LIN {X 0,Y 573.222,Z 156.084,A -85,B 0,C 180,E1 -2316.134,E2 -2316.134} C_VEL
LIN {X 0,Y 573.247,Z 156.08,A -85,B 0,C 180,E1 -2319.173,E2 -2319.173} C_VEL
LIN {X 0,Y 573.22,Z 156.083,A -85,B 0,C 180,E1 -2321.411,E2 -2321.411} C_VEL
LIN {X 0,Y 573.25,Z 156.076,A -85,B 0,C 180,E1 -2323.622,E2 -2323.622} C_VEL
LIN {X 0,Y 573.271,Z 156.075,A -85,B 0,C 180,E1 -2325.807,E2 -2325.807} C_VEL
LIN {X 0,Y 573.261,Z 156.075,A -85,B 0,C 180,E1 -2328.745,E2 -2328.745} C_VEL
LIN {X 0,Y 573.235,Z 156.083,A -85,B 0,C 180,E1 -2331.54,E2 -2331.54} C_VEL
LIN {X 0,Y 573.272,Z 156.074,A -85,B 0,C 180,E1 -2334.372,E2 -2334.372} C_VEL
LIN {X 0,Y 573.302,Z 156.07,A -85,B 0,C 180,E1 -2337.189,E2 -2337.189} C_VEL
LIN {X 0,Y 573.322,Z 156.073,A -85,B 0,C 180,E1 -2340,E2 -2340} C_VEL
LIN {X 0,Y 573.302,Z 156.07,A -85,B 0,C 180,E1 -2342.811,E2 -2342.811} C_VEL
LIN {X 0,Y 573.269,Z 156.075,A -85,B 0,C 180,E1 -2345.628,E2 -2345.628} C_VEL
LIN {X 0,Y 573.236,Z 156.083,A -85,B 0,C 180,E1 -2348.46,E2 -2348.46} C_VEL
LIN {X 0,Y 573.27,Z 156.073,A -85,B 0,C 180,E1 -2351.312,E2 -2351.312} C_VEL
LIN {X 0,Y 573.271,Z 156.075,A -85,B 0,C 180,E1 -2354.193,E2 -2354.193} C_VEL
LIN {X 0,Y 573.257,Z 156.081,A -85,B 0,C 180,E1 -2357.112,E2 -2357.112} C_VEL
LIN {X 0,Y 573.237,Z 156.079,A -85,B 0,C 180,E1 -2360.077,E2 -2360.077} C_VEL
LIN {X 0,Y 573.217,Z 156.086,A -85,B 0,C 180,E1 -2362.339,E2 -2362.339} C_VEL
LIN {X 0,Y 573.243,Z 156.077,A -85,B 0,C 180,E1 -2364.375,E2 -2364.375} C_VEL
LIN {X 0,Y 572.619,Z 156.154,A -85,B 0,C 180,E1 -2364.962,E2 -2364.962} C_VEL
LIN {X 0,Y 569.78,Z 156.514,A -85,B 0,C 180,E1 -2365.913,E2 -2365.913} C_VEL
LIN {X 0,Y 567.348,Z 156.82,A -85,B 0,C 180,E1 -2366.679,E2 -2366.679} C_VEL
LIN {X 0,Y 566.293,Z 156.949,A -85,B 0,C 180,E1 -2367.27,E2 -2367.27} C_VEL
LIN {X 0,Y 566.202,Z 156.958,A -85,B 0,C 180,E1 -2367.47,E2 -2367.47} C_VEL
LIN {X 0,Y 566.2,Z 156.955,A -85,B 0,C 180,E1 -2369.769,E2 -2369.769} C_VEL
LIN {X 0,Y 566.203,Z 156.96,A -85,B 0,C 180,E1 -2372.43,E2 -2372.43} C_VEL
LIN {X 0,Y 566.167,Z 156.959,A -85,B 0,C 180,E1 -2374.988,E2 -2374.988} C_VEL
LIN {X 0,Y 566.183,Z 156.961,A -85,B 0,C 180,E1 -2377.462,E2 -2377.462} C_VEL
LIN {X 0,Y 566.205,Z 156.953,A -85,B 0,C 180,E1 -2380.2,E2 -2380.2} C_VEL
LIN {X 0,Y 566.199,Z 156.958,A -85,B 0,C 180,E1 -2383.055,E2 -2383.055} C_VEL
LIN {X 0,Y 566.198,Z 156.959,A -85,B 0,C 180,E1 -2386.049,E2 -2386.049} C_VEL
LIN {X 0,Y 566.203,Z 156.956,A -85,B 0,C 180,E1 -2389.215,E2 -2389.215} C_VEL
LIN {X 0,Y 566.171,Z 156.962,A -85,B 0,C 180,E1 -2391.636,E2 -2391.636} C_VEL
LIN {X 0,Y 566.131,Z 156.965,A -85,B 0,C 180,E1 -2394.306,E2 -2394.306} C_VEL
LIN {X 0,Y 566.142,Z 157.825,A -85,B 0,C 180,E1 -2395.178,E2 -2395.178} C_VEL
LIN {X 0,Y 566.126,Z 162.015,A -85,B 0,C 180,E1 -2397.737,E2 -2397.737} C_VEL
LIN {X 0,Y 566.1,Z 166.291,A -85,B 0,C 180,E1 -2400.347,E2 -2400.347} C_VEL
LIN {X 0,Y 566.065,Z 170.142,A -85,B 0,C 180,E1 -2402.654,E2 -2402.654} C_VEL
LIN {X 0,Y 566.061,Z 174.191,A -85,B 0,C 180,E1 -2405.031,E2 -2405.031} C_VEL
LIN {X 0,Y 565.989,Z 178.243,A -85,B 0,C 180,E1 -2407.361,E2 -2407.361} C_VEL
LIN {X 0,Y 565.961,Z 182.275,A -85,B 0,C 180,E1 -2409.654,E2 -2409.654} C_VEL
LIN {X 0,Y 565.898,Z 186.291,A -85,B 0,C 180,E1 -2411.912,E2 -2411.912} C_VEL
LIN {X 0,Y 565.902,Z 191.779,A -85,B 0,C 180,E1 -2414.883,E2 -2414.883} C_VEL
LIN {X 0,Y 565.886,Z 196.532,A -85,B 0,C 180,E1 -2417.402,E2 -2417.402} C_VEL
LIN {X 0,Y 566.916,Z 203.459,A -85,B 0,C 180,E1 -2417.584,E2 -2417.584} C_VEL
LIN {X 0,Y 566.783,Z 216.489,A -85,B 0,C 180,E1 -2417.968,E2 -2417.968} C_VEL
LIN {X 0,Y 566.608,Z 229.064,A -85,B 0,C 180,E1 -2418.49,E2 -2418.49} C_VEL
LIN {X 0,Y 566.519,Z 240.338,A -85,B 0,C 180,E1 -2419.114,E2 -2419.114} C_VEL
LIN {X 0,Y 566.397,Z 251.686,A -85,B 0,C 180,E1 -2419.906,E2 -2419.906} C_VEL
LIN {X 0,Y 566.255,Z 261.061,A -85,B 0,C 180,E1 -2420.715,E2 -2420.715} C_VEL
LIN {X 0,Y 566.158,Z 269.617,A -85,B 0,C 180,E1 -2421.613,E2 -2421.613} C_VEL
LIN {X 0,Y 566.063,Z 277.929,A -85,B 0,C 180,E1 -2422.689,E2 -2422.689} C_VEL
LIN {X 0,Y 565.988,Z 284.624,A -85,B 0,C 180,E1 -2423.763,E2 -2423.763} C_VEL
LIN {X 0,Y 565.877,Z 290.765,A -85,B 0,C 180,E1 -2425.013,E2 -2425.013} C_VEL
LIN {X 0,Y 565.926,Z 294.754,A -85,B 0,C 180,E1 -2426.084,E2 -2426.084} C_VEL
LIN {X 0,Y 565.877,Z 297.703,A -85,B 0,C 180,E1 -2427.153,E2 -2427.153} C_VEL
LIN {X 0,Y 565.841,Z 299.128,A -85,B 0,C 180,E1 -2427.865,E2 -2427.865} C_VEL
LIN {X 0,Y 565.841,Z 300.756,A -85,B 0,C 180,E1 -2429.289,E2 -2429.289} C_VEL
LIN {X 0,Y 565.839,Z 300.996,A -85,B 0,C 180,E1 -2430,E2 -2430} C_VEL
LIN {X 0,Y 565.841,Z 300.815,A -85,B 0,C 180,E1 -2430.712,E2 -2430.712} C_VEL
LIN {X 0,Y 565.841,Z 299.267,A -85,B 0,C 180,E1 -2432.136,E2 -2432.136} C_VEL
LIN {X 0,Y 565.878,Z 297.906,A -85,B 0,C 180,E1 -2432.848,E2 -2432.848} C_VEL
LIN {X 0,Y 565.926,Z 295.029,A -85,B 0,C 180,E1 -2433.917,E2 -2433.917} C_VEL
LIN {X 0,Y 565.878,Z 291.128,A -85,B 0,C 180,E1 -2434.988,E2 -2434.988} C_VEL
LIN {X 0,Y 565.991,Z 286.096,A -85,B 0,C 180,E1 -2436.059,E2 -2436.059} C_VEL
LIN {X 0,Y 566.031,Z 279.771,A -85,B 0,C 180,E1 -2437.133,E2 -2437.133} C_VEL
LIN {X 0,Y 566.128,Z 271.849,A -85,B 0,C 180,E1 -2438.208,E2 -2438.208} C_VEL
LIN {X 0,Y 566.249,Z 261.997,A -85,B 0,C 180,E1 -2439.285,E2 -2439.285} C_VEL
LIN {X 0,Y 566.401,Z 251.679,A -85,B 0,C 180,E1 -2440.185,E2 -2440.185} C_VEL
LIN {X 0,Y 566.499,Z 240.539,A -85,B 0,C 180,E1 -2440.964,E2 -2440.964} C_VEL
LIN {X 0,Y 566.63,Z 229.184,A -85,B 0,C 180,E1 -2441.593,E2 -2441.593} C_VEL
LIN {X 0,Y 566.8,Z 216.59,A -85,B 0,C 180,E1 -2442.119,E2 -2442.119} C_VEL
LIN {X 0,Y 566.924,Z 203.412,A -85,B 0,C 180,E1 -2442.507,E2 -2442.507} C_VEL
LIN {X 0,Y 565.888,Z 196.529,A -85,B 0,C 180,E1 -2442.69,E2 -2442.69} C_VEL
LIN {X 0,Y 565.893,Z 191.947,A -85,B 0,C 180,E1 -2445.118,E2 -2445.118} C_VEL
LIN {X 0,Y 565.896,Z 186.449,A -85,B 0,C 180,E1 -2448.088,E2 -2448.088} C_VEL
LIN {X 0,Y 565.96,Z 182.428,A -85,B 0,C 180,E1 -2450.347,E2 -2450.347} C_VEL
LIN {X 0,Y 566.015,Z 177.311,A -85,B 0,C 180,E1 -2453.244,E2 -2453.244} C_VEL
LIN {X 0,Y 566.035,Z 173,A -85,B 0,C 180,E1 -2455.758,E2 -2455.758} C_VEL
LIN {X 0,Y 566.085,Z 168.894,A -85,B 0,C 180,E1 -2458.179,E2 -2458.179} C_VEL
LIN {X 0,Y 566.108,Z 164.128,A -85,B 0,C 180,E1 -2461.062,E2 -2461.062} C_VEL
LIN {X 0,Y 566.151,Z 159.371,A -85,B 0,C 180,E1 -2463.96,E2 -2463.96} C_VEL
LIN {X 0,Y 566.159,Z 157.704,A -85,B 0,C 180,E1 -2464.986,E2 -2464.986} C_VEL
LIN {X 0,Y 566.115,Z 156.967,A -85,B 0,C 180,E1 -2465.696,E2 -2465.696} C_VEL
LIN {X 0,Y 566.182,Z 156.962,A -85,B 0,C 180,E1 -2468.554,E2 -2468.554} C_VEL
LIN {X 0,Y 566.161,Z 156.959,A -85,B 0,C 180,E1 -2471.141,E2 -2471.141} C_VEL
LIN {X 0,Y 566.199,Z 156.959,A -85,B 0,C 180,E1 -2474.036,E2 -2474.036} C_VEL
LIN {X 0,Y 566.203,Z 156.958,A -85,B 0,C 180,E1 -2477.083,E2 -2477.083} C_VEL
LIN {X 0,Y 566.214,Z 156.954,A -85,B 0,C 180,E1 -2480.314,E2 -2480.314} C_VEL
LIN {X 0,Y 566.186,Z 156.96,A -85,B 0,C 180,E1 -2482.601,E2 -2482.601} C_VEL
LIN {X 0,Y 566.183,Z 156.957,A -85,B 0,C 180,E1 -2485.18,E2 -2485.18} C_VEL
LIN {X 0,Y 566.232,Z 156.955,A -85,B 0,C 180,E1 -2487.743,E2 -2487.743} C_VEL
LIN {X 0,Y 566.205,Z 156.954,A -85,B 0,C 180,E1 -2490.328,E2 -2490.328} C_VEL
LIN {X 0,Y 566.212,Z 156.959,A -85,B 0,C 180,E1 -2492.661,E2 -2492.661} C_VEL
LIN {X 0,Y 566.238,Z 156.949,A -85,B 0,C 180,E1 -2495.039,E2 -2495.039} C_VEL
LIN {X 0,Y 566.185,Z 156.959,A -85,B 0,C 180,E1 -2498.137,E2 -2498.137} C_VEL
LIN {X 0,Y 566.231,Z 156.951,A -85,B 0,C 180,E1 -2500.614,E2 -2500.614} C_VEL
LIN {X 0,Y 566.216,Z 156.954,A -85,B 0,C 180,E1 -2503.412,E2 -2503.412} C_VEL
LIN {X 0,Y 566.198,Z 156.961,A -85,B 0,C 180,E1 -2506.359,E2 -2506.359} C_VEL
LIN {X 0,Y 566.236,Z 156.95,A -85,B 0,C 180,E1 -2508.675,E2 -2508.675} C_VEL
LIN {X 0,Y 566.193,Z 156.961,A -85,B 0,C 180,E1 -2511.434,E2 -2511.434} C_VEL
LIN {X 0,Y 566.233,Z 156.95,A -85,B 0,C 180,E1 -2514.301,E2 -2514.301} C_VEL
LIN {X 0,Y 566.269,Z 156.947,A -85,B 0,C 180,E1 -2517.154,E2 -2517.154} C_VEL
LIN {X 0,Y 566.293,Z 156.949,A -85,B 0,C 180,E1 -2520,E2 -2520} C_VEL
LIN {X 0,Y 566.271,Z 156.946,A -85,B 0,C 180,E1 -2522.846,E2 -2522.846} C_VEL
LIN {X 0,Y 566.241,Z 156.95,A -85,B 0,C 180,E1 -2525.698,E2 -2525.698} C_VEL
LIN {X 0,Y 566.189,Z 156.961,A -85,B 0,C 180,E1 -2528.566,E2 -2528.566} C_VEL
LIN {X 0,Y 566.243,Z 156.95,A -85,B 0,C 180,E1 -2531.454,E2 -2531.454} C_VEL
LIN {X 0,Y 566.236,Z 156.95,A -85,B 0,C 180,E1 -2534.507,E2 -2534.507} C_VEL
LIN {X 0,Y 566.2,Z 156.96,A -85,B 0,C 180,E1 -2537.332,E2 -2537.332} C_VEL
LIN {X 0,Y 566.206,Z 156.957,A -85,B 0,C 180,E1 -2540.337,E2 -2540.337} C_VEL
LIN {X 0,Y 566.166,Z 156.958,A -85,B 0,C 180,E1 -2543.28,E2 -2543.28} C_VEL
LIN {X 0,Y 566.207,Z 156.96,A -85,B 0,C 180,E1 -2545.749,E2 -2545.749} C_VEL
LIN {X 0,Y 566.204,Z 156.954,A -85,B 0,C 180,E1 -2548.202,E2 -2548.202} C_VEL
LIN {X 0,Y 566.193,Z 156.96,A -85,B 0,C 180,E1 -2551.077,E2 -2551.077} C_VEL
LIN {X 0,Y 566.212,Z 156.954,A -85,B 0,C 180,E1 -2553.734,E2 -2553.734} C_VEL
LIN {X 0,Y 566.145,Z 156.962,A -85,B 0,C 180,E1 -2556.574,E2 -2556.574} C_VEL
LIN {X 0,Y 566.205,Z 156.958,A -85,B 0,C 180,E1 -2559.275,E2 -2559.275} C_VEL
LIN {X 0,Y 566.19,Z 156.955,A -85,B 0,C 180,E1 -2562.09,E2 -2562.09} C_VEL
LIN {X 0,Y 566.17,Z 156.96,A -85,B 0,C 180,E1 -2565.036,E2 -2565.036} C_VEL
LIN {X 0,Y 566.19,Z 156.961,A -85,B 0,C 180,E1 -2567.91,E2 -2567.91} C_VEL
LIN {X 0,Y 566.206,Z 156.955,A -85,B 0,C 180,E1 -2570.726,E2 -2570.726} C_VEL
LIN {X 0,Y 566.203,Z 157.05,A -85,B 0,C 180,E1 -2573.481,E2 -2573.481} C_VEL
LIN {X 0,Y 566.594,Z 160.732,A -85,B 0,C 180,E1 -2574.951,E2 -2574.951} C_VEL
LIN {X 0,Y 566.468,Z 168.073,A -85,B 0,C 180,E1 -2577.759,E2 -2577.759} C_VEL
LIN {X 0,Y 566.419,Z 174.878,A -85,B 0,C 180,E1 -2580.29,E2 -2580.29} C_VEL
LIN {X 0,Y 566.308,Z 183.258,A -85,B 0,C 180,E1 -2583.321,E2 -2583.321} C_VEL
LIN {X 0,Y 566.224,Z 191.447,A -85,B 0,C 180,E1 -2586.21,E2 -2586.21} C_VEL
LIN {X 0,Y 566.162,Z 199.239,A -85,B 0,C 180,E1 -2588.9,E2 -2588.9} C_VEL
LIN {X 0,Y 566.083,Z 207.03,A -85,B 0,C 180,E1 -2591.543,E2 -2591.543} C_VEL
LIN {X 0,Y 566.024,Z 215.935,A -85,B 0,C 180,E1 -2594.517,E2 -2594.517} C_VEL
LIN {X 0,Y 565.976,Z 224.283,A -85,B 0,C 180,E1 -2597.267,E2 -2597.267} C_VEL
LIN {X 0,Y 565.964,Z 224.491,A -85,B 0,C 180,E1 -2597.335,E2 -2597.335} C_VEL
LIN {X 0,Y 566.944,Z 231.504,A -85,B 0,C 180,E1 -2597.494,E2 -2597.494} C_VEL
LIN {X 0,Y 566.824,Z 243.874,A -85,B 0,C 180,E1 -2597.832,E2 -2597.832} C_VEL
LIN {X 0,Y 566.64,Z 256.897,A -85,B 0,C 180,E1 -2598.346,E2 -2598.346} C_VEL
LIN {X 0,Y 566.528,Z 268.482,A -85,B 0,C 180,E1 -2598.955,E2 -2598.955} C_VEL
LIN {X 0,Y 566.432,Z 279.927,A -85,B 0,C 180,E1 -2599.726,E2 -2599.726} C_VEL
LIN {X 0,Y 566.282,Z 289.599,A -85,B 0,C 180,E1 -2600.535,E2 -2600.535} C_VEL
LIN {X 0,Y 566.181,Z 298.412,A -85,B 0,C 180,E1 -2601.433,E2 -2601.433} C_VEL
LIN {X 0,Y 566.056,Z 306.999,A -85,B 0,C 180,E1 -2602.509,E2 -2602.509} C_VEL
LIN {X 0,Y 565.965,Z 313.866,A -85,B 0,C 180,E1 -2603.583,E2 -2603.583} C_VEL
LIN {X 0,Y 565.937,Z 319.365,A -85,B 0,C 180,E1 -2604.656,E2 -2604.656} C_VEL
LIN {X 0,Y 565.959,Z 323.677,A -85,B 0,C 180,E1 -2605.727,E2 -2605.727} C_VEL
LIN {X 0,Y 565.927,Z 325.956,A -85,B 0,C 180,E1 -2606.44,E2 -2606.44} C_VEL
LIN {X 0,Y 565.878,Z 327.808,A -85,B 0,C 180,E1 -2607.152,E2 -2607.152} C_VEL
LIN {X 0,Y 565.841,Z 329.2,A -85,B 0,C 180,E1 -2607.864,E2 -2607.864} C_VEL
LIN {X 0,Y 565.841,Z 330.784,A -85,B 0,C 180,E1 -2609.288,E2 -2609.288} C_VEL
LIN {X 0,Y 565.839,Z 331,A -85,B 0,C 180,E1 -2610,E2 -2610} C_VEL
LIN {X 0,Y 565.846,Z 330.186,A -85,B 0,C 180,E1 -2611.423,E2 -2611.423} C_VEL
LIN {X 0,Y 565.841,Z 329.201,A -85,B 0,C 180,E1 -2612.135,E2 -2612.135} C_VEL
LIN {X 0,Y 565.878,Z 327.81,A -85,B 0,C 180,E1 -2612.847,E2 -2612.847} C_VEL
LIN {X 0,Y 565.926,Z 324.897,A -85,B 0,C 180,E1 -2613.916,E2 -2613.916} C_VEL
LIN {X 0,Y 565.878,Z 320.95,A -85,B 0,C 180,E1 -2614.987,E2 -2614.987} C_VEL
LIN {X 0,Y 566.002,Z 315.867,A -85,B 0,C 180,E1 -2616.058,E2 -2616.058} C_VEL
LIN {X 0,Y 566.04,Z 309.471,A -85,B 0,C 180,E1 -2617.132,E2 -2617.132} C_VEL
LIN {X 0,Y 566.133,Z 301.48,A -85,B 0,C 180,E1 -2618.207,E2 -2618.207} C_VEL
LIN {X 0,Y 566.229,Z 293.339,A -85,B 0,C 180,E1 -2619.105,E2 -2619.105} C_VEL
LIN {X 0,Y 566.336,Z 283.405,A -85,B 0,C 180,E1 -2620.005,E2 -2620.005} C_VEL
LIN {X 0,Y 566.469,Z 272.332,A -85,B 0,C 180,E1 -2620.805,E2 -2620.805} C_VEL
LIN {X 0,Y 566.608,Z 259.955,A -85,B 0,C 180,E1 -2621.51,E2 -2621.51} C_VEL
LIN {X 0,Y 566.746,Z 247.773,A -85,B 0,C 180,E1 -2622.033,E2 -2622.033} C_VEL
LIN {X 0,Y 566.906,Z 234.359,A -85,B 0,C 180,E1 -2622.439,E2 -2622.439} C_VEL
LIN {X 0,Y 566.632,Z 228.828,A -85,B 0,C 180,E1 -2622.567,E2 -2622.567} C_VEL
LIN {X 0,Y 565.963,Z 224.492,A -85,B 0,C 180,E1 -2622.665,E2 -2622.665} C_VEL
LIN {X 0,Y 566.019,Z 217.049,A -85,B 0,C 180,E1 -2625.114,E2 -2625.114} C_VEL
LIN {X 0,Y 566.065,Z 208.144,A -85,B 0,C 180,E1 -2628.082,E2 -2628.082} C_VEL
LIN {X 0,Y 566.145,Z 200.353,A -85,B 0,C 180,E1 -2630.719,E2 -2630.719} C_VEL
LIN {X 0,Y 566.205,Z 192.562,A -85,B 0,C 180,E1 -2633.403,E2 -2633.403} C_VEL
LIN {X 0,Y 566.294,Z 184.77,A -85,B 0,C 180,E1 -2636.14,E2 -2636.14} C_VEL
LIN {X 0,Y 566.383,Z 176.979,A -85,B 0,C 180,E1 -2638.942,E2 -2638.942} C_VEL
LIN {X 0,Y 566.477,Z 169.187,A -85,B 0,C 180,E1 -2641.821,E2 -2641.821} C_VEL
LIN {X 0,Y 566.567,Z 161.396,A -85,B 0,C 180,E1 -2644.792,E2 -2644.792} C_VEL
LIN {X 0,Y 566.225,Z 157.187,A -85,B 0,C 180,E1 -2646.466,E2 -2646.466} C_VEL
LIN {X 0,Y 566.201,Z 156.961,A -85,B 0,C 180,E1 -2646.569,E2 -2646.569} C_VEL
LIN {X 0,Y 566.208,Z 156.955,A -85,B 0,C 180,E1 -2649.685,E2 -2649.685} C_VEL
LIN {X 0,Y 566.208,Z 156.96,A -85,B 0,C 180,E1 -2652.087,E2 -2652.087} C_VEL
LIN {X 0,Y 566.168,Z 156.961,A -85,B 0,C 180,E1 -2655.036,E2 -2655.036} C_VEL
LIN {X 0,Y 566.188,Z 156.956,A -85,B 0,C 180,E1 -2657.91,E2 -2657.91} C_VEL
LIN {X 0,Y 566.206,Z 156.958,A -85,B 0,C 180,E1 -2660.725,E2 -2660.725} C_VEL
LIN {X 0,Y 566.143,Z 156.962,A -85,B 0,C 180,E1 -2663.426,E2 -2663.426} C_VEL
LIN {X 0,Y 566.209,Z 156.954,A -85,B 0,C 180,E1 -2666.266,E2 -2666.266} C_VEL
LIN {X 0,Y 566.194,Z 156.959,A -85,B 0,C 180,E1 -2668.922,E2 -2668.922} C_VEL
LIN {X 0,Y 566.21,Z 156.953,A -85,B 0,C 180,E1 -2671.857,E2 -2671.857} C_VEL
LIN {X 0,Y 566.211,Z 156.96,A -85,B 0,C 180,E1 -2674.251,E2 -2674.251} C_VEL
LIN {X 0,Y 566.164,Z 156.958,A -85,B 0,C 180,E1 -2676.72,E2 -2676.72} C_VEL
LIN {X 0,Y 566.204,Z 156.958,A -85,B 0,C 180,E1 -2679.662,E2 -2679.662} C_VEL
LIN {X 0,Y 566.198,Z 156.959,A -85,B 0,C 180,E1 -2682.668,E2 -2682.668} C_VEL
LIN {X 0,Y 566.232,Z 156.951,A -85,B 0,C 180,E1 -2685.627,E2 -2685.627} C_VEL
LIN {X 0,Y 566.232,Z 156.95,A -85,B 0,C 180,E1 -2688.675,E2 -2688.675} C_VEL
LIN {X 0,Y 566.189,Z 156.962,A -85,B 0,C 180,E1 -2691.434,E2 -2691.434} C_VEL
LIN {X 0,Y 566.238,Z 156.95,A -85,B 0,C 180,E1 -2694.301,E2 -2694.301} C_VEL
LIN {X 0,Y 566.275,Z 156.947,A -85,B 0,C 180,E1 -2697.866,E2 -2697.866} C_VEL
LIN {X 0,Y 566.301,Z 156.942,A -85,B 0,C 180,E1 -2700.711,E2 -2700.711} C_VEL
LIN {X 0,Y 566.269,Z 156.947,A -85,B 0,C 180,E1 -2702.846,E2 -2702.846} C_VEL
LIN {X 0,Y 566.236,Z 156.95,A -85,B 0,C 180,E1 -2705.699,E2 -2705.699} C_VEL
LIN {X 0,Y 566.19,Z 156.962,A -85,B 0,C 180,E1 -2708.566,E2 -2708.566} C_VEL
LIN {X 0,Y 566.24,Z 156.95,A -85,B 0,C 180,E1 -2711.454,E2 -2711.454} C_VEL
LIN {X 0,Y 566.233,Z 156.95,A -85,B 0,C 180,E1 -2714.507,E2 -2714.507} C_VEL
LIN {X 0,Y 566.198,Z 156.959,A -85,B 0,C 180,E1 -2717.332,E2 -2717.332} C_VEL
LIN {X 0,Y 566.203,Z 156.958,A -85,B 0,C 180,E1 -2720.338,E2 -2720.338} C_VEL
LIN {X 0,Y 566.164,Z 156.958,A -85,B 0,C 180,E1 -2723.28,E2 -2723.28} C_VEL
LIN {X 0,Y 566.211,Z 156.959,A -85,B 0,C 180,E1 -2725.749,E2 -2725.749} C_VEL
LIN {X 0,Y 566.202,Z 156.958,A -85,B 0,C 180,E1 -2727.47,E2 -2727.47} C_VEL
LIN {X 0,Y 565.521,Z 157.04,A -85,B 0,C 180,E1 -2728.064,E2 -2728.064} C_VEL
LIN {X 0,Y 562.656,Z 157.401,A -85,B 0,C 180,E1 -2729.027,E2 -2729.027} C_VEL
LIN {X 0,Y 560.247,Z 157.698,A -85,B 0,C 180,E1 -2729.803,E2 -2729.803} C_VEL
LIN {X 0,Y 559.22,Z 157.826,A -85,B 0,C 180,E1 -2730.402,E2 -2730.402} C_VEL
LIN {X 0,Y 559.139,Z 157.835,A -85,B 0,C 180,E1 -2730.604,E2 -2730.604} C_VEL
LIN {X 0,Y 559.156,Z 157.837,A -85,B 0,C 180,E1 -2732.715,E2 -2732.715} C_VEL
LIN {X 0,Y 559.115,Z 157.837,A -85,B 0,C 180,E1 -2735.325,E2 -2735.325} C_VEL
LIN {X 0,Y 559.121,Z 157.838,A -85,B 0,C 180,E1 -2738.019,E2 -2738.019} C_VEL
LIN {X 0,Y 559.155,Z 157.834,A -85,B 0,C 180,E1 -2740.813,E2 -2740.813} C_VEL
LIN {X 0,Y 559.138,Z 157.834,A -85,B 0,C 180,E1 -2743.734,E2 -2743.734} C_VEL
LIN {X 0,Y 559.146,Z 157.834,A -85,B 0,C 180,E1 -2746.804,E2 -2746.804} C_VEL
LIN {X 0,Y 559.155,Z 157.834,A -85,B 0,C 180,E1 -2749.188,E2 -2749.188} C_VEL
LIN {X 0,Y 559.121,Z 157.837,A -85,B 0,C 180,E1 -2751.982,E2 -2751.982} C_VEL
LIN {X 0,Y 559.054,Z 157.882,A -85,B 0,C 180,E1 -2754.671,E2 -2754.671} C_VEL
LIN {X 0,Y 559.057,Z 162.259,A -85,B 0,C 180,E1 -2757.381,E2 -2757.381} C_VEL
LIN {X 0,Y 559.053,Z 166.761,A -85,B 0,C 180,E1 -2760.16,E2 -2760.16} C_VEL
LIN {X 0,Y 558.994,Z 171.604,A -85,B 0,C 180,E1 -2763.089,E2 -2763.089} C_VEL
LIN {X 0,Y 558.955,Z 175.655,A -85,B 0,C 180,E1 -2765.486,E2 -2765.486} C_VEL
LIN {X 0,Y 558.929,Z 180.876,A -85,B 0,C 180,E1 -2768.51,E2 -2768.51} C_VEL
LIN {X 0,Y 558.89,Z 185.109,A -85,B 0,C 180,E1 -2770.917,E2 -2770.917} C_VEL
LIN {X 0,Y 558.788,Z 190.462,A -85,B 0,C 180,E1 -2773.937,E2 -2773.937} C_VEL
LIN {X 0,Y 558.781,Z 194.545,A -85,B 0,C 180,E1 -2776.174,E2 -2776.174} C_VEL
LIN {X 0,Y 558.817,Z 196.533,A -85,B 0,C 180,E1 -2777.24,E2 -2777.24} C_VEL
LIN {X 0,Y 560.002,Z 204.395,A -85,B 0,C 180,E1 -2777.451,E2 -2777.451} C_VEL
LIN {X 0,Y 559.846,Z 216.89,A -85,B 0,C 180,E1 -2777.83,E2 -2777.83} C_VEL
LIN {X 0,Y 559.665,Z 228.866,A -85,B 0,C 180,E1 -2778.335,E2 -2778.335} C_VEL
LIN {X 0,Y 559.531,Z 240.553,A -85,B 0,C 180,E1 -2778.989,E2 -2778.989} C_VEL
LIN {X 0,Y 559.393,Z 251.692,A -85,B 0,C 180,E1 -2779.778,E2 -2779.778} C_VEL
LIN {X 0,Y 559.239,Z 261.068,A -85,B 0,C 180,E1 -2780.598,E2 -2780.598} C_VEL
LIN {X 0,Y 559.129,Z 269.623,A -85,B 0,C 180,E1 -2781.507,E2 -2781.507} C_VEL
LIN {X 0,Y 558.988,Z 277.932,A -85,B 0,C 180,E1 -2782.596,E2 -2782.596} C_VEL
LIN {X 0,Y 558.89,Z 284.414,A -85,B 0,C 180,E1 -2783.645,E2 -2783.645} C_VEL
LIN {X 0,Y 558.869,Z 289.165,A -85,B 0,C 180,E1 -2784.588,E2 -2784.588} C_VEL
LIN {X 0,Y 558.868,Z 293.523,A -85,B 0,C 180,E1 -2785.673,E2 -2785.673} C_VEL
LIN {X 0,Y 558.836,Z 295.829,A -85,B 0,C 180,E1 -2786.395,E2 -2786.395} C_VEL
LIN {X 0,Y 558.799,Z 297.705,A -85,B 0,C 180,E1 -2787.117,E2 -2787.117} C_VEL
LIN {X 0,Y 558.747,Z 299.128,A -85,B 0,C 180,E1 -2787.838,E2 -2787.838} C_VEL
LIN {X 0,Y 558.741,Z 300.757,A -85,B 0,C 180,E1 -2789.279,E2 -2789.279} C_VEL
LIN {X 0,Y 558.74,Z 300.996,A -85,B 0,C 180,E1 -2790,E2 -2790} C_VEL
LIN {X 0,Y 558.741,Z 300.815,A -85,B 0,C 180,E1 -2790.721,E2 -2790.721} C_VEL
LIN {X 0,Y 558.747,Z 299.265,A -85,B 0,C 180,E1 -2792.163,E2 -2792.163} C_VEL
LIN {X 0,Y 558.8,Z 297.904,A -85,B 0,C 180,E1 -2792.884,E2 -2792.884} C_VEL
LIN {X 0,Y 558.844,Z 295.027,A -85,B 0,C 180,E1 -2793.966,E2 -2793.966} C_VEL
LIN {X 0,Y 558.798,Z 291.126,A -85,B 0,C 180,E1 -2795.051,E2 -2795.051} C_VEL
LIN {X 0,Y 558.911,Z 286.094,A -85,B 0,C 180,E1 -2796.136,E2 -2796.136} C_VEL
LIN {X 0,Y 558.973,Z 279.767,A -85,B 0,C 180,E1 -2797.223,E2 -2797.223} C_VEL
LIN {X 0,Y 559.091,Z 271.844,A -85,B 0,C 180,E1 -2798.312,E2 -2798.312} C_VEL
LIN {X 0,Y 559.223,Z 261.99,A -85,B 0,C 180,E1 -2799.403,E2 -2799.403} C_VEL
LIN {X 0,Y 559.399,Z 251.669,A -85,B 0,C 180,E1 -2800.313,E2 -2800.313} C_VEL
LIN {X 0,Y 559.504,Z 240.822,A -85,B 0,C 180,E1 -2801.084,E2 -2801.084} C_VEL
LIN {X 0,Y 559.639,Z 230.269,A -85,B 0,C 180,E1 -2801.683,E2 -2801.683} C_VEL
LIN {X 0,Y 559.838,Z 217.741,A -85,B 0,C 180,E1 -2802.23,E2 -2802.23} C_VEL
LIN {X 0,Y 559.988,Z 204.304,A -85,B 0,C 180,E1 -2802.641,E2 -2802.641} C_VEL
LIN {X 0,Y 558.786,Z 196.528,A -85,B 0,C 180,E1 -2802.854,E2 -2802.854} C_VEL
LIN {X 0,Y 558.812,Z 191.964,A -85,B 0,C 180,E1 -2805.314,E2 -2805.314} C_VEL
LIN {X 0,Y 558.825,Z 186.593,A -85,B 0,C 180,E1 -2808.325,E2 -2808.325} C_VEL
LIN {X 0,Y 558.882,Z 182.561,A -85,B 0,C 180,E1 -2810.616,E2 -2810.616} C_VEL
LIN {X 0,Y 558.942,Z 177.747,A -85,B 0,C 180,E1 -2813.381,E2 -2813.381} C_VEL
LIN {X 0,Y 558.966,Z 173.106,A -85,B 0,C 180,E1 -2816.108,E2 -2816.108} C_VEL
LIN {X 0,Y 559.035,Z 169.048,A -85,B 0,C 180,E1 -2818.537,E2 -2818.537} C_VEL
LIN {X 0,Y 559.072,Z 164.601,A -85,B 0,C 180,E1 -2821.26,E2 -2821.26} C_VEL
LIN {X 0,Y 559.107,Z 159.435,A -85,B 0,C 180,E1 -2824.448,E2 -2824.448} C_VEL
LIN {X 0,Y 559.08,Z 158.027,A -85,B 0,C 180,E1 -2825.328,E2 -2825.328} C_VEL
LIN {X 0,Y 559.118,Z 157.837,A -85,B 0,C 180,E1 -2827.637,E2 -2827.637} C_VEL
LIN {X 0,Y 559.157,Z 157.833,A -85,B 0,C 180,E1 -2829.941,E2 -2829.941} C_VEL
LIN {X 0,Y 559.158,Z 157.832,A -85,B 0,C 180,E1 -2832.744,E2 -2832.744} C_VEL
LIN {X 0,Y 559.151,Z 157.836,A -85,B 0,C 180,E1 -2835.761,E2 -2835.761} C_VEL
LIN {X 0,Y 559.164,Z 157.83,A -85,B 0,C 180,E1 -2838.23,E2 -2838.23} C_VEL
LIN {X 0,Y 559.171,Z 157.831,A -85,B 0,C 180,E1 -2841.192,E2 -2841.192} C_VEL
LIN {X 0,Y 559.115,Z 157.84,A -85,B 0,C 180,E1 -2843.787,E2 -2843.787} C_VEL
LIN {X 0,Y 559.146,Z 157.834,A -85,B 0,C 180,E1 -2846.424,E2 -2846.424} C_VEL
LIN {X 0,Y 559.157,Z 157.836,A -85,B 0,C 180,E1 -2848.981,E2 -2848.981} C_VEL
LIN {X 0,Y 559.17,Z 157.83,A -85,B 0,C 180,E1 -2851.619,E2 -2851.619} C_VEL
LIN {X 0,Y 559.182,Z 157.829,A -85,B 0,C 180,E1 -2853.903,E2 -2853.903} C_VEL
LIN {X 0,Y 559.137,Z 157.835,A -85,B 0,C 180,E1 -2856.572,E2 -2856.572} C_VEL
LIN {X 0,Y 559.174,Z 157.834,A -85,B 0,C 180,E1 -2859.395,E2 -2859.395} C_VEL
LIN {X 0,Y 559.139,Z 157.836,A -85,B 0,C 180,E1 -2861.685,E2 -2861.685} C_VEL
LIN {X 0,Y 559.167,Z 157.831,A -85,B 0,C 180,E1 -2863.948,E2 -2863.948} C_VEL
LIN {X 0,Y 559.173,Z 157.835,A -85,B 0,C 180,E1 -2866.184,E2 -2866.184} C_VEL
LIN {X 0,Y 559.194,Z 157.827,A -85,B 0,C 180,E1 -2869.133,E2 -2869.133} C_VEL
LIN {X 0,Y 559.138,Z 157.834,A -85,B 0,C 180,E1 -2872.053,E2 -2872.053} C_VEL
LIN {X 0,Y 559.24,Z 157.827,A -85,B 0,C 180,E1 -2874.953,E2 -2874.953} C_VEL
LIN {X 0,Y 559.245,Z 157.822,A -85,B 0,C 180,E1 -2877.839,E2 -2877.839} C_VEL
LIN {X 0,Y 559.274,Z 157.818,A -85,B 0,C 180,E1 -2880.72,E2 -2880.72} C_VEL
LIN {X 0,Y 559.237,Z 157.822,A -85,B 0,C 180,E1 -2882.881,E2 -2882.881} C_VEL
LIN {X 0,Y 559.209,Z 157.825,A -85,B 0,C 180,E1 -2885.77,E2 -2885.77} C_VEL
LIN {X 0,Y 559.156,Z 157.838,A -85,B 0,C 180,E1 -2888.675,E2 -2888.675} C_VEL
LIN {X 0,Y 559.206,Z 157.827,A -85,B 0,C 180,E1 -2891.6,E2 -2891.6} C_VEL
LIN {X 0,Y 559.202,Z 157.826,A -85,B 0,C 180,E1 -2894.596,E2 -2894.596} C_VEL
LIN {X 0,Y 559.143,Z 157.836,A -85,B 0,C 180,E1 -2897.557,E2 -2897.557} C_VEL
LIN {X 0,Y 559.166,Z 157.83,A -85,B 0,C 180,E1 -2899.838,E2 -2899.838} C_VEL
LIN {X 0,Y 559.137,Z 157.839,A -85,B 0,C 180,E1 -2902.153,E2 -2902.153} C_VEL
LIN {X 0,Y 559.175,Z 157.831,A -85,B 0,C 180,E1 -2905.298,E2 -2905.298} C_VEL
LIN {X 0,Y 559.169,Z 157.83,A -85,B 0,C 180,E1 -2908.381,E2 -2908.381} C_VEL
LIN {X 0,Y 559.148,Z 157.835,A -85,B 0,C 180,E1 -2911.273,E2 -2911.273} C_VEL
LIN {X 0,Y 559.165,Z 157.833,A -85,B 0,C 180,E1 -2913.949,E2 -2913.949} C_VEL
LIN {X 0,Y 559.112,Z 157.837,A -85,B 0,C 180,E1 -2917.111,E2 -2917.111} C_VEL
LIN {X 0,Y 559.157,Z 157.832,A -85,B 0,C 180,E1 -2919.941,E2 -2919.941} C_VEL
LIN {X 0,Y 559.158,Z 157.836,A -85,B 0,C 180,E1 -2922.744,E2 -2922.744} C_VEL
LIN {X 0,Y 559.151,Z 157.834,A -85,B 0,C 180,E1 -2925.761,E2 -2925.761} C_VEL
LIN {X 0,Y 559.164,Z 157.835,A -85,B 0,C 180,E1 -2928.23,E2 -2928.23} C_VEL
LIN {X 0,Y 559.168,Z 157.836,A -85,B 0,C 180,E1 -2931.193,E2 -2931.193} C_VEL
LIN {X 0,Y 559.19,Z 157.999,A -85,B 0,C 180,E1 -2933.341,E2 -2933.341} C_VEL
LIN {X 0,Y 559.588,Z 162.52,A -85,B 0,C 180,E1 -2935.155,E2 -2935.155} C_VEL
LIN {X 0,Y 559.47,Z 170.299,A -85,B 0,C 180,E1 -2938.157,E2 -2938.157} C_VEL
LIN {X 0,Y 559.428,Z 176.978,A -85,B 0,C 180,E1 -2940.663,E2 -2940.663} C_VEL
LIN {X 0,Y 559.275,Z 184.835,A -85,B 0,C 180,E1 -2943.53,E2 -2943.53} C_VEL
LIN {X 0,Y 559.167,Z 193.358,A -85,B 0,C 180,E1 -2946.566,E2 -2946.566} C_VEL
LIN {X 0,Y 559.097,Z 201.465,A -85,B 0,C 180,E1 -2949.392,E2 -2949.392} C_VEL
LIN {X 0,Y 559.01,Z 209.256,A -85,B 0,C 180,E1 -2952.06,E2 -2952.06} C_VEL
LIN {X 0,Y 558.943,Z 217.048,A -85,B 0,C 180,E1 -2954.689,E2 -2954.689} C_VEL
LIN {X 0,Y 558.906,Z 224.491,A -85,B 0,C 180,E1 -2957.172,E2 -2957.172} C_VEL
LIN {X 0,Y 560.004,Z 232.518,A -85,B 0,C 180,E1 -2957.359,E2 -2957.359} C_VEL
LIN {X 0,Y 559.883,Z 245.304,A -85,B 0,C 180,E1 -2957.729,E2 -2957.729} C_VEL
LIN {X 0,Y 559.682,Z 258.23,A -85,B 0,C 180,E1 -2958.261,E2 -2958.261} C_VEL
LIN {X 0,Y 559.549,Z 268.95,A -85,B 0,C 180,E1 -2958.843,E2 -2958.843} C_VEL
LIN {X 0,Y 559.42,Z 279.926,A -85,B 0,C 180,E1 -2959.596,E2 -2959.596} C_VEL
LIN {X 0,Y 559.243,Z 289.599,A -85,B 0,C 180,E1 -2960.415,E2 -2960.415} C_VEL
LIN {X 0,Y 559.127,Z 298.412,A -85,B 0,C 180,E1 -2961.325,E2 -2961.325} C_VEL
LIN {X 0,Y 558.996,Z 306.999,A -85,B 0,C 180,E1 -2962.414,E2 -2962.414} C_VEL
LIN {X 0,Y 558.885,Z 314.687,A -85,B 0,C 180,E1 -2963.649,E2 -2963.649} C_VEL
LIN {X 0,Y 558.869,Z 319.365,A -85,B 0,C 180,E1 -2964.588,E2 -2964.588} C_VEL
LIN {X 0,Y 558.868,Z 323.677,A -85,B 0,C 180,E1 -2965.673,E2 -2965.673} C_VEL
LIN {X 0,Y 558.836,Z 325.956,A -85,B 0,C 180,E1 -2966.395,E2 -2966.395} C_VEL
LIN {X 0,Y 558.799,Z 327.808,A -85,B 0,C 180,E1 -2967.116,E2 -2967.116} C_VEL
LIN {X 0,Y 558.746,Z 329.199,A -85,B 0,C 180,E1 -2967.837,E2 -2967.837} C_VEL
LIN {X 0,Y 558.741,Z 330.784,A -85,B 0,C 180,E1 -2969.279,E2 -2969.279} C_VEL
LIN {X 0,Y 558.74,Z 331,A -85,B 0,C 180,E1 -2970,E2 -2970} C_VEL
LIN {X 0,Y 558.745,Z 330.186,A -85,B 0,C 180,E1 -2971.441,E2 -2971.441} C_VEL
LIN {X 0,Y 558.746,Z 329.201,A -85,B 0,C 180,E1 -2972.162,E2 -2972.162} C_VEL
LIN {X 0,Y 558.799,Z 327.81,A -85,B 0,C 180,E1 -2972.883,E2 -2972.883} C_VEL
LIN {X 0,Y 558.844,Z 324.896,A -85,B 0,C 180,E1 -2973.966,E2 -2973.966} C_VEL
LIN {X 0,Y 558.798,Z 320.95,A -85,B 0,C 180,E1 -2975.051,E2 -2975.051} C_VEL
LIN {X 0,Y 558.921,Z 315.867,A -85,B 0,C 180,E1 -2976.135,E2 -2976.135} C_VEL
LIN {X 0,Y 558.977,Z 309.471,A -85,B 0,C 180,E1 -2977.223,E2 -2977.223} C_VEL
LIN {X 0,Y 559.099,Z 301.48,A -85,B 0,C 180,E1 -2978.311,E2 -2978.311} C_VEL
LIN {X 0,Y 559.194,Z 293.339,A -85,B 0,C 180,E1 -2979.221,E2 -2979.221} C_VEL
LIN {X 0,Y 559.346,Z 283.404,A -85,B 0,C 180,E1 -2980.131,E2 -2980.131} C_VEL
LIN {X 0,Y 559.474,Z 272.441,A -85,B 0,C 180,E1 -2980.935,E2 -2980.935} C_VEL
LIN {X 0,Y 559.635,Z 260.827,A -85,B 0,C 180,E1 -2981.61,E2 -2981.61} C_VEL
LIN {X 0,Y 559.786,Z 248.993,A -85,B 0,C 180,E1 -2982.139,E2 -2982.139} C_VEL
LIN {X 0,Y 559.968,Z 236.187,A -85,B 0,C 180,E1 -2982.549,E2 -2982.549} C_VEL
LIN {X 0,Y 559.833,Z 230.38,A -85,B 0,C 180,E1 -2982.691,E2 -2982.691} C_VEL
LIN {X 0,Y 558.905,Z 224.492,A -85,B 0,C 180,E1 -2982.827,E2 -2982.827} C_VEL
LIN {X 0,Y 558.942,Z 217.049,A -85,B 0,C 180,E1 -2985.31,E2 -2985.31} C_VEL
LIN {X 0,Y 559.01,Z 209.257,A -85,B 0,C 180,E1 -2987.94,E2 -2987.94} C_VEL
LIN {X 0,Y 559.101,Z 201.466,A -85,B 0,C 180,E1 -2990.607,E2 -2990.607} C_VEL
LIN {X 0,Y 559.166,Z 193.359,A -85,B 0,C 180,E1 -2993.434,E2 -2993.434} C_VEL
LIN {X 0,Y 559.275,Z 184.836,A -85,B 0,C 180,E1 -2996.47,E2 -2996.47} C_VEL
LIN {X 0,Y 559.427,Z 176.979,A -85,B 0,C 180,E1 -2999.337,E2 -2999.337} C_VEL
LIN {X 0,Y 559.483,Z 169.187,A -85,B 0,C 180,E1 -3002.267,E2 -3002.267} C_VEL
LIN {X 0,Y 559.585,Z 161.388,A -85,B 0,C 180,E1 -3005.291,E2 -3005.291} C_VEL
LIN {X 0,Y 559.157,Z 157.838,A -85,B 0,C 180,E1 -3006.75,E2 -3006.75} C_VEL
LIN {X 0,Y 559.174,Z 157.833,A -85,B 0,C 180,E1 -3009.866,E2 -3009.866} C_VEL
LIN {X 0,Y 559.16,Z 157.832,A -85,B 0,C 180,E1 -3012.743,E2 -3012.743} C_VEL
LIN {X 0,Y 559.148,Z 157.836,A -85,B 0,C 180,E1 -3015.761,E2 -3015.761} C_VEL
LIN {X 0,Y 559.161,Z 157.831,A -85,B 0,C 180,E1 -3018.229,E2 -3018.229} C_VEL
LIN {X 0,Y 559.167,Z 157.83,A -85,B 0,C 180,E1 -3021.192,E2 -3021.192} C_VEL
LIN {X 0,Y 559.113,Z 157.841,A -85,B 0,C 180,E1 -3023.787,E2 -3023.787} C_VEL
LIN {X 0,Y 559.16,Z 157.832,A -85,B 0,C 180,E1 -3026.425,E2 -3026.425} C_VEL
LIN {X 0,Y 559.159,Z 157.837,A -85,B 0,C 180,E1 -3028.981,E2 -3028.981} C_VEL
LIN {X 0,Y 559.167,Z 157.831,A -85,B 0,C 180,E1 -3031.619,E2 -3031.619} C_VEL
LIN {X 0,Y 559.178,Z 157.831,A -85,B 0,C 180,E1 -3033.903,E2 -3033.903} C_VEL
LIN {X 0,Y 559.134,Z 157.834,A -85,B 0,C 180,E1 -3036.572,E2 -3036.572} C_VEL
LIN {X 0,Y 559.173,Z 157.835,A -85,B 0,C 180,E1 -3039.395,E2 -3039.395} C_VEL
LIN {X 0,Y 559.14,Z 157.835,A -85,B 0,C 180,E1 -3041.685,E2 -3041.685} C_VEL
LIN {X 0,Y 559.166,Z 157.831,A -85,B 0,C 180,E1 -3043.948,E2 -3043.948} C_VEL
LIN {X 0,Y 559.17,Z 157.836,A -85,B 0,C 180,E1 -3046.184,E2 -3046.184} C_VEL
LIN {X 0,Y 559.19,Z 157.828,A -85,B 0,C 180,E1 -3049.133,E2 -3049.133} C_VEL
LIN {X 0,Y 559.135,Z 157.834,A -85,B 0,C 180,E1 -3052.053,E2 -3052.053} C_VEL
LIN {X 0,Y 559.243,Z 157.827,A -85,B 0,C 180,E1 -3054.953,E2 -3054.953} C_VEL
LIN {X 0,Y 559.247,Z 157.822,A -85,B 0,C 180,E1 -3057.839,E2 -3057.839} C_VEL
LIN {X 0,Y 559.271,Z 157.818,A -85,B 0,C 180,E1 -3060.72,E2 -3060.72} C_VEL
LIN {X 0,Y 559.235,Z 157.823,A -85,B 0,C 180,E1 -3062.881,E2 -3062.881} C_VEL
LIN {X 0,Y 559.204,Z 157.826,A -85,B 0,C 180,E1 -3065.77,E2 -3065.77} C_VEL
LIN {X 0,Y 559.156,Z 157.836,A -85,B 0,C 180,E1 -3068.675,E2 -3068.675} C_VEL
LIN {X 0,Y 559.203,Z 157.828,A -85,B 0,C 180,E1 -3071.601,E2 -3071.601} C_VEL
LIN {X 0,Y 559.198,Z 157.827,A -85,B 0,C 180,E1 -3074.596,E2 -3074.596} C_VEL
LIN {X 0,Y 559.157,Z 157.834,A -85,B 0,C 180,E1 -3077.557,E2 -3077.557} C_VEL
LIN {X 0,Y 559.163,Z 157.831,A -85,B 0,C 180,E1 -3079.838,E2 -3079.838} C_VEL
LIN {X 0,Y 559.131,Z 157.841,A -85,B 0,C 180,E1 -3082.153,E2 -3082.153} C_VEL
LIN {X 0,Y 559.174,Z 157.831,A -85,B 0,C 180,E1 -3085.298,E2 -3085.298} C_VEL
LIN {X 0,Y 559.179,Z 157.832,A -85,B 0,C 180,E1 -3087.712,E2 -3087.712} C_VEL
LIN {X 0,Y 559.139,Z 157.835,A -85,B 0,C 180,E1 -3090.604,E2 -3090.604} C_VEL
LIN {X 0,Y 558.477,Z 157.921,A -85,B 0,C 180,E1 -3091.206,E2 -3091.206} C_VEL
LIN {X 0,Y 555.615,Z 158.276,A -85,B 0,C 180,E1 -3092.182,E2 -3092.182} C_VEL
LIN {X 0,Y 553.202,Z 158.576,A -85,B 0,C 180,E1 -3092.967,E2 -3092.967} C_VEL
LIN {X 0,Y 552.18,Z 158.702,A -85,B 0,C 180,E1 -3093.574,E2 -3093.574} C_VEL
LIN {X 0,Y 552.105,Z 158.712,A -85,B 0,C 180,E1 -3093.779,E2 -3093.779} C_VEL
LIN {X 0,Y 552.066,Z 158.715,A -85,B 0,C 180,E1 -3096.75,E2 -3096.75} C_VEL
LIN {X 0,Y 552.126,Z 158.712,A -85,B 0,C 180,E1 -3099.528,E2 -3099.528} C_VEL
LIN {X 0,Y 552.129,Z 158.709,A -85,B 0,C 180,E1 -3102.426,E2 -3102.426} C_VEL
LIN {X 0,Y 552.098,Z 158.711,A -85,B 0,C 180,E1 -3105.563,E2 -3105.563} C_VEL
LIN {X 0,Y 552.12,Z 158.709,A -85,B 0,C 180,E1 -3108.554,E2 -3108.554} C_VEL
LIN {X 0,Y 552.109,Z 158.715,A -85,B 0,C 180,E1 -3111.411,E2 -3111.411} C_VEL
LIN {X 0,Y 552.047,Z 158.718,A -85,B 0,C 180,E1 -3114.154,E2 -3114.154} C_VEL
LIN {X 0,Y 552.006,Z 158.727,A -85,B 0,C 180,E1 -3114.571,E2 -3114.571} C_VEL
LIN {X 0,Y 552.007,Z 162.748,A -85,B 0,C 180,E1 -3117.172,E2 -3117.172} C_VEL
LIN {X 0,Y 552.002,Z 167.647,A -85,B 0,C 180,E1 -3120.229,E2 -3120.229} C_VEL
LIN {X 0,Y 551.946,Z 172.248,A -85,B 0,C 180,E1 -3123.04,E2 -3123.04} C_VEL
LIN {X 0,Y 551.879,Z 177.135,A -85,B 0,C 180,E1 -3125.952,E2 -3125.952} C_VEL
LIN {X 0,Y 551.873,Z 181.271,A -85,B 0,C 180,E1 -3128.38,E2 -3128.38} C_VEL
LIN {X 0,Y 551.764,Z 186.598,A -85,B 0,C 180,E1 -3131.432,E2 -3131.432} C_VEL
LIN {X 0,Y 551.721,Z 190.635,A -85,B 0,C 180,E1 -3133.726,E2 -3133.726} C_VEL
LIN {X 0,Y 551.699,Z 194.662,A -85,B 0,C 180,E1 -3135.993,E2 -3135.993} C_VEL
LIN {X 0,Y 551.704,Z 196.589,A -85,B 0,C 180,E1 -3137.072,E2 -3137.072} C_VEL
LIN {X 0,Y 553.059,Z 205.337,A -85,B 0,C 180,E1 -3137.315,E2 -3137.315} C_VEL
LIN {X 0,Y 552.897,Z 217.814,A -85,B 0,C 180,E1 -3137.707,E2 -3137.707} C_VEL
LIN {X 0,Y 552.668,Z 230.32,A -85,B 0,C 180,E1 -3138.261,E2 -3138.261} C_VEL
LIN {X 0,Y 552.512,Z 241.821,A -85,B 0,C 180,E1 -3138.93,E2 -3138.93} C_VEL
LIN {X 0,Y 552.346,Z 252.863,A -85,B 0,C 180,E1 -3139.739,E2 -3139.739} C_VEL
LIN {X 0,Y 552.175,Z 262.901,A -85,B 0,C 180,E1 -3140.661,E2 -3140.661} C_VEL
LIN {X 0,Y 552.007,Z 272.601,A -85,B 0,C 180,E1 -3141.765,E2 -3141.765} C_VEL
LIN {X 0,Y 551.895,Z 280.462,A -85,B 0,C 180,E1 -3142.886,E2 -3142.886} C_VEL
LIN {X 0,Y 551.868,Z 287.458,A -85,B 0,C 180,E1 -3144.153,E2 -3144.153} C_VEL
LIN {X 0,Y 551.725,Z 292.198,A -85,B 0,C 180,E1 -3145.251,E2 -3145.251} C_VEL
LIN {X 0,Y 551.751,Z 295.83,A -85,B 0,C 180,E1 -3146.349,E2 -3146.349} C_VEL
LIN {X 0,Y 551.723,Z 297.707,A -85,B 0,C 180,E1 -3147.08,E2 -3147.08} C_VEL
LIN {X 0,Y 551.657,Z 299.128,A -85,B 0,C 180,E1 -3147.81,E2 -3147.81} C_VEL
LIN {X 0,Y 551.642,Z 300.757,A -85,B 0,C 180,E1 -3149.27,E2 -3149.27} C_VEL
LIN {X 0,Y 551.641,Z 300.996,A -85,B 0,C 180,E1 -3150,E2 -3150} C_VEL
LIN {X 0,Y 551.641,Z 300.815,A -85,B 0,C 180,E1 -3150.73,E2 -3150.73} C_VEL
LIN {X 0,Y 551.657,Z 299.263,A -85,B 0,C 180,E1 -3152.191,E2 -3152.191} C_VEL
LIN {X 0,Y 551.724,Z 297.902,A -85,B 0,C 180,E1 -3152.921,E2 -3152.921} C_VEL
LIN {X 0,Y 551.764,Z 295.025,A -85,B 0,C 180,E1 -3154.017,E2 -3154.017} C_VEL
LIN {X 0,Y 551.723,Z 291.124,A -85,B 0,C 180,E1 -3155.116,E2 -3155.116} C_VEL
LIN {X 0,Y 551.811,Z 285.391,A -85,B 0,C 180,E1 -3156.349,E2 -3156.349} C_VEL
LIN {X 0,Y 551.925,Z 278.535,A -85,B 0,C 180,E1 -3157.5,E2 -3157.5} C_VEL
LIN {X 0,Y 552.063,Z 270.353,A -85,B 0,C 180,E1 -3158.603,E2 -3158.603} C_VEL
LIN {X 0,Y 552.196,Z 261.984,A -85,B 0,C 180,E1 -3159.524,E2 -3159.524} C_VEL
LIN {X 0,Y 552.38,Z 251.66,A -85,B 0,C 180,E1 -3160.446,E2 -3160.446} C_VEL
LIN {X 0,Y 552.534,Z 240.049,A -85,B 0,C 180,E1 -3161.275,E2 -3161.275} C_VEL
LIN {X 0,Y 552.744,Z 228.445,A -85,B 0,C 180,E1 -3161.924,E2 -3161.924} C_VEL
LIN {X 0,Y 552.922,Z 216.425,A -85,B 0,C 180,E1 -3162.432,E2 -3162.432} C_VEL
LIN {X 0,Y 552.939,Z 203.948,A -85,B 0,C 180,E1 -3162.814,E2 -3162.814} C_VEL
LIN {X 0,Y 551.679,Z 196.58,A -85,B 0,C 180,E1 -3163.022,E2 -3163.022} C_VEL
LIN {X 0,Y 551.728,Z 192.138,A -85,B 0,C 180,E1 -3165.516,E2 -3165.516} C_VEL
LIN {X 0,Y 551.757,Z 188.076,A -85,B 0,C 180,E1 -3167.8,E2 -3167.8} C_VEL
LIN {X 0,Y 551.8,Z 184.049,A -85,B 0,C 180,E1 -3170.114,E2 -3170.114} C_VEL
LIN {X 0,Y 551.846,Z 179.988,A -85,B 0,C 180,E1 -3172.462,E2 -3172.462} C_VEL
LIN {X 0,Y 551.916,Z 175.173,A -85,B 0,C 180,E1 -3175.297,E2 -3175.297} C_VEL
LIN {X 0,Y 551.954,Z 170.508,A -85,B 0,C 180,E1 -3178.107,E2 -3178.107} C_VEL
LIN {X 0,Y 551.985,Z 166.432,A -85,B 0,C 180,E1 -3180.617,E2 -3180.617} C_VEL
LIN {X 0,Y 552.018,Z 162.309,A -85,B 0,C 180,E1 -3183.193,E2 -3183.193} C_VEL
LIN {X 0,Y 552.019,Z 158.741,A -85,B 0,C 180,E1 -3185.431,E2 -3185.431} C_VEL
LIN {X 0,Y 552.076,Z 158.714,A -85,B 0,C 180,E1 -3187.882,E2 -3187.882} C_VEL
LIN {X 0,Y 552.094,Z 158.717,A -85,B 0,C 180,E1 -3190.483,E2 -3190.483} C_VEL
LIN {X 0,Y 552.094,Z 158.714,A -85,B 0,C 180,E1 -3193.481,E2 -3193.481} C_VEL
LIN {X 0,Y 552.109,Z 158.71,A -85,B 0,C 180,E1 -3196.576,E2 -3196.576} C_VEL
LIN {X 0,Y 552.11,Z 158.71,A -85,B 0,C 180,E1 -3199.519,E2 -3199.519} C_VEL
LIN {X 0,Y 552.082,Z 158.718,A -85,B 0,C 180,E1 -3202.335,E2 -3202.335} C_VEL
LIN {X 0,Y 552.074,Z 158.714,A -85,B 0,C 180,E1 -3205.05,E2 -3205.05} C_VEL
LIN {X 0,Y 552.116,Z 158.714,A -85,B 0,C 180,E1 -3207.681,E2 -3207.681} C_VEL
LIN {X 0,Y 552.113,Z 158.709,A -85,B 0,C 180,E1 -3210.235,E2 -3210.235} C_VEL
LIN {X 0,Y 552.14,Z 158.708,A -85,B 0,C 180,E1 -3213,E2 -3213} C_VEL
LIN {X 0,Y 552.114,Z 158.708,A -85,B 0,C 180,E1 -3215.161,E2 -3215.161} C_VEL
LIN {X 0,Y 552.127,Z 158.708,A -85,B 0,C 180,E1 -3218.337,E2 -3218.337} C_VEL
LIN {X 0,Y 552.151,Z 158.706,A -85,B 0,C 180,E1 -3220.674,E2 -3220.674} C_VEL
LIN {X 0,Y 552.117,Z 158.709,A -85,B 0,C 180,E1 -3223.737,E2 -3223.737} C_VEL
LIN {X 0,Y 552.137,Z 158.709,A -85,B 0,C 180,E1 -3226.004,E2 -3226.004} C_VEL
LIN {X 0,Y 552.162,Z 158.703,A -85,B 0,C 180,E1 -3228.993,E2 -3228.993} C_VEL
LIN {X 0,Y 552.108,Z 158.711,A -85,B 0,C 180,E1 -3231.951,E2 -3231.951} C_VEL
LIN {X 0,Y 552.215,Z 158.702,A -85,B 0,C 180,E1 -3234.889,E2 -3234.889} C_VEL
LIN {X 0,Y 552.218,Z 158.697,A -85,B 0,C 180,E1 -3237.812,E2 -3237.812} C_VEL
LIN {X 0,Y 552.244,Z 158.693,A -85,B 0,C 180,E1 -3240.729,E2 -3240.729} C_VEL
LIN {X 0,Y 552.204,Z 158.699,A -85,B 0,C 180,E1 -3242.918,E2 -3242.918} C_VEL
LIN {X 0,Y 552.178,Z 158.701,A -85,B 0,C 180,E1 -3245.844,E2 -3245.844} C_VEL
LIN {X 0,Y 552.129,Z 158.712,A -85,B 0,C 180,E1 -3248.786,E2 -3248.786} C_VEL
LIN {X 0,Y 552.163,Z 158.706,A -85,B 0,C 180,E1 -3251.75,E2 -3251.75} C_VEL
LIN {X 0,Y 552.138,Z 158.707,A -85,B 0,C 180,E1 -3254.748,E2 -3254.748} C_VEL
LIN {X 0,Y 552.1,Z 158.712,A -85,B 0,C 180,E1 -3257.789,E2 -3257.789} C_VEL
LIN {X 0,Y 552.126,Z 158.709,A -85,B 0,C 180,E1 -3260.101,E2 -3260.101} C_VEL
LIN {X 0,Y 552.088,Z 158.717,A -85,B 0,C 180,E1 -3262.451,E2 -3262.451} C_VEL
LIN {X 0,Y 552.138,Z 158.708,A -85,B 0,C 180,E1 -3265.346,E2 -3265.346} C_VEL
LIN {X 0,Y 552.103,Z 158.711,A -85,B 0,C 180,E1 -3268.099,E2 -3268.099} C_VEL
LIN {X 0,Y 552.104,Z 158.714,A -85,B 0,C 180,E1 -3270.609,E2 -3270.609} C_VEL
LIN {X 0,Y 552.116,Z 158.71,A -85,B 0,C 180,E1 -3273.186,E2 -3273.186} C_VEL
LIN {X 0,Y 552.07,Z 158.719,A -85,B 0,C 180,E1 -3275.845,E2 -3275.845} C_VEL
LIN {X 0,Y 552.115,Z 158.71,A -85,B 0,C 180,E1 -3279.06,E2 -3279.06} C_VEL
LIN {X 0,Y 552.122,Z 158.711,A -85,B 0,C 180,E1 -3281.446,E2 -3281.446} C_VEL
LIN {X 0,Y 552.092,Z 158.718,A -85,B 0,C 180,E1 -3284.531,E2 -3284.531} C_VEL
LIN {X 0,Y 552.131,Z 158.709,A -85,B 0,C 180,E1 -3287.585,E2 -3287.585} C_VEL
LIN {X 0,Y 552.126,Z 158.709,A -85,B 0,C 180,E1 -3290.472,E2 -3290.472} C_VEL
LIN {X 0,Y 552.13,Z 158.816,A -85,B 0,C 180,E1 -3293.141,E2 -3293.141} C_VEL
LIN {X 0,Y 552.577,Z 162.085,A -85,B 0,C 180,E1 -3294.488,E2 -3294.488} C_VEL
LIN {X 0,Y 552.524,Z 168.705,A -85,B 0,C 180,E1 -3297.088,E2 -3297.088} C_VEL
LIN {X 0,Y 552.389,Z 176.05,A -85,B 0,C 180,E1 -3299.901,E2 -3299.901} C_VEL
LIN {X 0,Y 552.272,Z 184.307,A -85,B 0,C 180,E1 -3302.974,E2 -3302.974} C_VEL
LIN {X 0,Y 552.159,Z 192.561,A -85,B 0,C 180,E1 -3305.964,E2 -3305.964} C_VEL
LIN {X 0,Y 552.058,Z 200.352,A -85,B 0,C 180,E1 -3308.726,E2 -3308.726} C_VEL
LIN {X 0,Y 551.949,Z 208.143,A -85,B 0,C 180,E1 -3311.438,E2 -3311.438} C_VEL
LIN {X 0,Y 551.9,Z 217.048,A -85,B 0,C 180,E1 -3314.489,E2 -3314.489} C_VEL
LIN {X 0,Y 551.812,Z 224.491,A -85,B 0,C 180,E1 -3317.004,E2 -3317.004} C_VEL
LIN {X 0,Y 553.086,Z 233.433,A -85,B 0,C 180,E1 -3317.222,E2 -3317.222} C_VEL
LIN {X 0,Y 552.935,Z 246.47,A -85,B 0,C 180,E1 -3317.614,E2 -3317.614} C_VEL
LIN {X 0,Y 552.722,Z 257.482,A -85,B 0,C 180,E1 -3318.075,E2 -3318.075} C_VEL
LIN {X 0,Y 552.56,Z 269.382,A -85,B 0,C 180,E1 -3318.726,E2 -3318.726} C_VEL
LIN {X 0,Y 552.412,Z 281.095,A -85,B 0,C 180,E1 -3319.555,E2 -3319.555} C_VEL
LIN {X 0,Y 552.201,Z 291.536,A -85,B 0,C 180,E1 -3320.476,E2 -3320.476} C_VEL
LIN {X 0,Y 552.082,Z 299.989,A -85,B 0,C 180,E1 -3321.397,E2 -3321.397} C_VEL
LIN {X 0,Y 551.927,Z 308.236,A -85,B 0,C 180,E1 -3322.5,E2 -3322.5} C_VEL
LIN {X 0,Y 551.821,Z 315.208,A -85,B 0,C 180,E1 -3323.662,E2 -3323.662} C_VEL
LIN {X 0,Y 551.723,Z 320.949,A -85,B 0,C 180,E1 -3324.884,E2 -3324.884} C_VEL
LIN {X 0,Y 551.764,Z 324.895,A -85,B 0,C 180,E1 -3325.983,E2 -3325.983} C_VEL
LIN {X 0,Y 551.723,Z 327.808,A -85,B 0,C 180,E1 -3327.079,E2 -3327.079} C_VEL
LIN {X 0,Y 551.657,Z 329.199,A -85,B 0,C 180,E1 -3327.809,E2 -3327.809} C_VEL
LIN {X 0,Y 551.641,Z 330.785,A -85,B 0,C 180,E1 -3329.27,E2 -3329.27} C_VEL
LIN {X 0,Y 551.64,Z 331,A -85,B 0,C 180,E1 -3330,E2 -3330} C_VEL
LIN {X 0,Y 551.645,Z 330.186,A -85,B 0,C 180,E1 -3331.46,E2 -3331.46} C_VEL
LIN {X 0,Y 551.657,Z 329.2,A -85,B 0,C 180,E1 -3332.19,E2 -3332.19} C_VEL
LIN {X 0,Y 551.723,Z 327.81,A -85,B 0,C 180,E1 -3332.92,E2 -3332.92} C_VEL
LIN {X 0,Y 551.764,Z 324.896,A -85,B 0,C 180,E1 -3334.017,E2 -3334.017} C_VEL
LIN {X 0,Y 551.723,Z 320.95,A -85,B 0,C 180,E1 -3335.116,E2 -3335.116} C_VEL
LIN {X 0,Y 551.825,Z 315.19,A -85,B 0,C 180,E1 -3336.341,E2 -3336.341} C_VEL
LIN {X 0,Y 551.926,Z 308.239,A -85,B 0,C 180,E1 -3337.499,E2 -3337.499} C_VEL
LIN {X 0,Y 552.082,Z 299.992,A -85,B 0,C 180,E1 -3338.602,E2 -3338.602} C_VEL
LIN {X 0,Y 552.199,Z 291.54,A -85,B 0,C 180,E1 -3339.523,E2 -3339.523} C_VEL
LIN {X 0,Y 552.412,Z 281.099,A -85,B 0,C 180,E1 -3340.445,E2 -3340.445} C_VEL
LIN {X 0,Y 552.552,Z 270.421,A -85,B 0,C 180,E1 -3341.206,E2 -3341.206} C_VEL
LIN {X 0,Y 552.699,Z 259.416,A -85,B 0,C 180,E1 -3341.832,E2 -3341.832} C_VEL
LIN {X 0,Y 552.897,Z 247.77,A -85,B 0,C 180,E1 -3342.339,E2 -3342.339} C_VEL
LIN {X 0,Y 553.066,Z 234.358,A -85,B 0,C 180,E1 -3342.755,E2 -3342.755} C_VEL
LIN {X 0,Y 552.572,Z 229.112,A -85,B 0,C 180,E1 -3342.886,E2 -3342.886} C_VEL
LIN {X 0,Y 551.812,Z 224.492,A -85,B 0,C 180,E1 -3342.995,E2 -3342.995} C_VEL
LIN {X 0,Y 551.896,Z 215.936,A -85,B 0,C 180,E1 -3345.89,E2 -3345.89} C_VEL
LIN {X 0,Y 551.993,Z 207.031,A -85,B 0,C 180,E1 -3348.945,E2 -3348.945} C_VEL
LIN {X 0,Y 552.075,Z 199.215,A -85,B 0,C 180,E1 -3351.673,E2 -3351.673} C_VEL
LIN {X 0,Y 552.18,Z 191.449,A -85,B 0,C 180,E1 -3354.434,E2 -3354.434} C_VEL
LIN {X 0,Y 552.3,Z 183.657,A -85,B 0,C 180,E1 -3357.264,E2 -3357.264} C_VEL
LIN {X 0,Y 552.389,Z 176.051,A -85,B 0,C 180,E1 -3360.099,E2 -3360.099} C_VEL
LIN {X 0,Y 552.522,Z 168.706,A -85,B 0,C 180,E1 -3362.911,E2 -3362.911} C_VEL
LIN {X 0,Y 552.582,Z 162.094,A -85,B 0,C 180,E1 -3365.513,E2 -3365.513} C_VEL
LIN {X 0,Y 552.12,Z 158.715,A -85,B 0,C 180,E1 -3366.973,E2 -3366.973} C_VEL
LIN {X 0,Y 552.124,Z 158.709,A -85,B 0,C 180,E1 -3369.527,E2 -3369.527} C_VEL
LIN {X 0,Y 552.13,Z 158.709,A -85,B 0,C 180,E1 -3372.425,E2 -3372.425} C_VEL
LIN {X 0,Y 552.093,Z 158.716,A -85,B 0,C 180,E1 -3375.562,E2 -3375.562} C_VEL
LIN {X 0,Y 552.119,Z 158.711,A -85,B 0,C 180,E1 -3378.554,E2 -3378.554} C_VEL
LIN {X 0,Y 552.109,Z 158.709,A -85,B 0,C 180,E1 -3381.41,E2 -3381.41} C_VEL
LIN {X 0,Y 552.063,Z 158.716,A -85,B 0,C 180,E1 -3384.562,E2 -3384.562} C_VEL
LIN {X 0,Y 552.114,Z 158.713,A -85,B 0,C 180,E1 -3387.153,E2 -3387.153} C_VEL
LIN {X 0,Y 552.119,Z 158.709,A -85,B 0,C 180,E1 -3389.948,E2 -3389.948} C_VEL
LIN {X 0,Y 552.137,Z 158.708,A -85,B 0,C 180,E1 -3393,E2 -3393} C_VEL
LIN {X 0,Y 552.11,Z 158.709,A -85,B 0,C 180,E1 -3395.161,E2 -3395.161} C_VEL
LIN {X 0,Y 552.124,Z 158.708,A -85,B 0,C 180,E1 -3398.337,E2 -3398.337} C_VEL
LIN {X 0,Y 552.149,Z 158.706,A -85,B 0,C 180,E1 -3400.674,E2 -3400.674} C_VEL
LIN {X 0,Y 552.115,Z 158.709,A -85,B 0,C 180,E1 -3403.737,E2 -3403.737} C_VEL
LIN {X 0,Y 552.134,Z 158.71,A -85,B 0,C 180,E1 -3406.004,E2 -3406.004} C_VEL
LIN {X 0,Y 552.158,Z 158.704,A -85,B 0,C 180,E1 -3408.993,E2 -3408.993} C_VEL
LIN {X 0,Y 552.105,Z 158.71,A -85,B 0,C 180,E1 -3411.951,E2 -3411.951} C_VEL
LIN {X 0,Y 552.217,Z 158.703,A -85,B 0,C 180,E1 -3414.889,E2 -3414.889} C_VEL
LIN {X 0,Y 552.219,Z 158.698,A -85,B 0,C 180,E1 -3417.812,E2 -3417.812} C_VEL
LIN {X 0,Y 552.241,Z 158.694,A -85,B 0,C 180,E1 -3420.729,E2 -3420.729} C_VEL
LIN {X 0,Y 552.202,Z 158.7,A -85,B 0,C 180,E1 -3422.918,E2 -3422.918} C_VEL
LIN {X 0,Y 552.174,Z 158.702,A -85,B 0,C 180,E1 -3425.844,E2 -3425.844} C_VEL
LIN {X 0,Y 552.129,Z 158.71,A -85,B 0,C 180,E1 -3428.786,E2 -3428.786} C_VEL
LIN {X 0,Y 552.161,Z 158.707,A -85,B 0,C 180,E1 -3431.751,E2 -3431.751} C_VEL
LIN {X 0,Y 552.135,Z 158.707,A -85,B 0,C 180,E1 -3434.749,E2 -3434.749} C_VEL
LIN {X 0,Y 552.107,Z 158.711,A -85,B 0,C 180,E1 -3437.789,E2 -3437.789} C_VEL
LIN {X 0,Y 552.123,Z 158.71,A -85,B 0,C 180,E1 -3440.102,E2 -3440.102} C_VEL
LIN {X 0,Y 552.083,Z 158.717,A -85,B 0,C 180,E1 -3442.451,E2 -3442.451} C_VEL
LIN {X 0,Y 552.154,Z 158.706,A -85,B 0,C 180,E1 -3445.351,E2 -3445.351} C_VEL
LIN {X 0,Y 552.118,Z 158.709,A -85,B 0,C 180,E1 -3448.098,E2 -3448.098} C_VEL
LIN {X 0,Y 552.102,Z 158.715,A -85,B 0,C 180,E1 -3450.609,E2 -3450.609} C_VEL
LIN {X 0,Y 552.114,Z 158.71,A -85,B 0,C 180,E1 -3453.186,E2 -3453.186} C_VEL
LIN {X 0,Y 552.105,Z 158.712,A -85,B 0,C 180,E1 -3453.779,E2 -3453.779} C_VEL
LIN {X 0,Y 551.455,Z 158.797,A -85,B 0,C 180,E1 -3454.388,E2 -3454.388} C_VEL
LIN {X 0,Y 548.586,Z 159.152,A -85,B 0,C 180,E1 -3455.376,E2 -3455.376} C_VEL
LIN {X 0,Y 546.147,Z 159.456,A -85,B 0,C 180,E1 -3456.171,E2 -3456.171} C_VEL
LIN {X 0,Y 545.097,Z 159.584,A -85,B 0,C 180,E1 -3456.785,E2 -3456.785} C_VEL
LIN {X 0,Y 545.012,Z 159.594,A -85,B 0,C 180,E1 -3456.993,E2 -3456.993} C_VEL
LIN {X 0,Y 545.097,Z 159.589,A -85,B 0,C 180,E1 -3459.324,E2 -3459.324} C_VEL
LIN {X 0,Y 545.077,Z 159.585,A -85,B 0,C 180,E1 -3462.103,E2 -3462.103} C_VEL
LIN {X 0,Y 545.062,Z 159.588,A -85,B 0,C 180,E1 -3465.168,E2 -3465.168} C_VEL
LIN {X 0,Y 545.077,Z 159.59,A -85,B 0,C 180,E1 -3467.897,E2 -3467.897} C_VEL
LIN {X 0,Y 545.074,Z 159.587,A -85,B 0,C 180,E1 -3470.818,E2 -3470.818} C_VEL
LIN {X 0,Y 545.024,Z 159.594,A -85,B 0,C 180,E1 -3473.619,E2 -3473.619} C_VEL
LIN {X 0,Y 544.974,Z 159.603,A -85,B 0,C 180,E1 -3474.527,E2 -3474.527} C_VEL
LIN {X 0,Y 544.967,Z 163.621,A -85,B 0,C 180,E1 -3477.205,E2 -3477.205} C_VEL
LIN {X 0,Y 544.934,Z 167.741,A -85,B 0,C 180,E1 -3479.803,E2 -3479.803} C_VEL
LIN {X 0,Y 544.873,Z 171.822,A -85,B 0,C 180,E1 -3482.333,E2 -3482.333} C_VEL
LIN {X 0,Y 544.882,Z 175.889,A -85,B 0,C 180,E1 -3484.809,E2 -3484.809} C_VEL
LIN {X 0,Y 544.802,Z 181.318,A -85,B 0,C 180,E1 -3488.031,E2 -3488.031} C_VEL
LIN {X 0,Y 544.737,Z 185.378,A -85,B 0,C 180,E1 -3490.401,E2 -3490.401} C_VEL
LIN {X 0,Y 544.657,Z 190.804,A -85,B 0,C 180,E1 -3493.508,E2 -3493.508} C_VEL
LIN {X 0,Y 544.632,Z 194.845,A -85,B 0,C 180,E1 -3495.808,E2 -3495.808} C_VEL
LIN {X 0,Y 544.62,Z 196.778,A -85,B 0,C 180,E1 -3496.901,E2 -3496.901} C_VEL
LIN {X 0,Y 546.128,Z 206.486,A -85,B 0,C 180,E1 -3497.175,E2 -3497.175} C_VEL
LIN {X 0,Y 545.95,Z 219.226,A -85,B 0,C 180,E1 -3497.595,E2 -3497.595} C_VEL
LIN {X 0,Y 545.72,Z 231.659,A -85,B 0,C 180,E1 -3498.171,E2 -3498.171} C_VEL
LIN {X 0,Y 545.521,Z 243.057,A -85,B 0,C 180,E1 -3498.858,E2 -3498.858} C_VEL
LIN {X 0,Y 545.333,Z 254.055,A -85,B 0,C 180,E1 -3499.699,E2 -3499.699} C_VEL
LIN {X 0,Y 545.122,Z 264.744,A -85,B 0,C 180,E1 -3500.726,E2 -3500.726} C_VEL
LIN {X 0,Y 544.975,Z 272.626,A -85,B 0,C 180,E1 -3501.658,E2 -3501.658} C_VEL
LIN {X 0,Y 544.829,Z 280.353,A -85,B 0,C 180,E1 -3502.775,E2 -3502.775} C_VEL
LIN {X 0,Y 544.778,Z 287.46,A -85,B 0,C 180,E1 -3504.076,E2 -3504.076} C_VEL
LIN {X 0,Y 544.628,Z 292.2,A -85,B 0,C 180,E1 -3505.189,E2 -3505.189} C_VEL
LIN {X 0,Y 544.669,Z 295.831,A -85,B 0,C 180,E1 -3506.301,E2 -3506.301} C_VEL
LIN {X 0,Y 544.65,Z 297.709,A -85,B 0,C 180,E1 -3507.042,E2 -3507.042} C_VEL
LIN {X 0,Y 544.572,Z 299.128,A -85,B 0,C 180,E1 -3507.781,E2 -3507.781} C_VEL
LIN {X 0,Y 544.542,Z 300.757,A -85,B 0,C 180,E1 -3509.261,E2 -3509.261} C_VEL
LIN {X 0,Y 544.542,Z 300.996,A -85,B 0,C 180,E1 -3510,E2 -3510} C_VEL
LIN {X 0,Y 544.542,Z 300.814,A -85,B 0,C 180,E1 -3510.74,E2 -3510.74} C_VEL
LIN {X 0,Y 544.572,Z 299.261,A -85,B 0,C 180,E1 -3512.219,E2 -3512.219} C_VEL
LIN {X 0,Y 544.651,Z 297.9,A -85,B 0,C 180,E1 -3512.959,E2 -3512.959} C_VEL
LIN {X 0,Y 544.684,Z 295.023,A -85,B 0,C 180,E1 -3514.07,E2 -3514.07} C_VEL
LIN {X 0,Y 544.653,Z 291.121,A -85,B 0,C 180,E1 -3515.182,E2 -3515.182} C_VEL
LIN {X 0,Y 544.725,Z 285.895,A -85,B 0,C 180,E1 -3516.336,E2 -3516.336} C_VEL
LIN {X 0,Y 544.859,Z 278.531,A -85,B 0,C 180,E1 -3517.598,E2 -3517.598} C_VEL
LIN {X 0,Y 545.016,Z 270.38,A -85,B 0,C 180,E1 -3518.715,E2 -3518.715} C_VEL
LIN {X 0,Y 545.185,Z 262.046,A -85,B 0,C 180,E1 -3519.647,E2 -3519.647} C_VEL
LIN {X 0,Y 545.372,Z 251.759,A -85,B 0,C 180,E1 -3520.582,E2 -3520.582} C_VEL
LIN {X 0,Y 545.558,Z 240.593,A -85,B 0,C 180,E1 -3521.394,E2 -3521.394} C_VEL
LIN {X 0,Y 545.763,Z 230.418,A -85,B 0,C 180,E1 -3521.985,E2 -3521.985} C_VEL
LIN {X 0,Y 545.981,Z 217.908,A -85,B 0,C 180,E1 -3522.546,E2 -3522.546} C_VEL
LIN {X 0,Y 546.058,Z 205.051,A -85,B 0,C 180,E1 -3522.955,E2 -3522.955} C_VEL
LIN {X 0,Y 544.602,Z 196.752,A -85,B 0,C 180,E1 -3523.194,E2 -3523.194} C_VEL
LIN {X 0,Y 544.637,Z 192.31,A -85,B 0,C 180,E1 -3525.723,E2 -3525.723} C_VEL
LIN {X 0,Y 544.674,Z 188.22,A -85,B 0,C 180,E1 -3528.04,E2 -3528.04} C_VEL
LIN {X 0,Y 544.747,Z 184.181,A -85,B 0,C 180,E1 -3530.386,E2 -3530.386} C_VEL
LIN {X 0,Y 544.795,Z 180.116,A -85,B 0,C 180,E1 -3532.769,E2 -3532.769} C_VEL
LIN {X 0,Y 544.846,Z 175.606,A -85,B 0,C 180,E1 -3535.453,E2 -3535.453} C_VEL
LIN {X 0,Y 544.943,Z 170.611,A -85,B 0,C 180,E1 -3538.501,E2 -3538.501} C_VEL
LIN {X 0,Y 544.938,Z 166.52,A -85,B 0,C 180,E1 -3541.056,E2 -3541.056} C_VEL
LIN {X 0,Y 544.996,Z 162.376,A -85,B 0,C 180,E1 -3543.677,E2 -3543.677} C_VEL
LIN {X 0,Y 544.986,Z 159.602,A -85,B 0,C 180,E1 -3545.472,E2 -3545.472} C_VEL
LIN {X 0,Y 545.026,Z 159.594,A -85,B 0,C 180,E1 -3548.24,E2 -3548.24} C_VEL
LIN {X 0,Y 545.031,Z 159.592,A -85,B 0,C 180,E1 -3551.119,E2 -3551.119} C_VEL
LIN {X 0,Y 545.053,Z 159.592,A -85,B 0,C 180,E1 -3554.13,E2 -3554.13} C_VEL
LIN {X 0,Y 545.065,Z 159.592,A -85,B 0,C 180,E1 -3557.303,E2 -3557.303} C_VEL
LIN {X 0,Y 545.066,Z 159.586,A -85,B 0,C 180,E1 -3559.857,E2 -3559.857} C_VEL
LIN {X 0,Y 545.018,Z 159.596,A -85,B 0,C 180,E1 -3562.694,E2 -3562.694} C_VEL
LIN {X 0,Y 545.054,Z 159.593,A -85,B 0,C 180,E1 -3565.611,E2 -3565.611} C_VEL
LIN {X 0,Y 545.059,Z 159.588,A -85,B 0,C 180,E1 -3568.321,E2 -3568.321} C_VEL
LIN {X 0,Y 545.091,Z 159.587,A -85,B 0,C 180,E1 -3571.252,E2 -3571.252} C_VEL
LIN {X 0,Y 545.081,Z 159.587,A -85,B 0,C 180,E1 -3573.999,E2 -3573.999} C_VEL
LIN {X 0,Y 545.078,Z 159.588,A -85,B 0,C 180,E1 -3576.44,E2 -3576.44} C_VEL
LIN {X 0,Y 545.091,Z 159.59,A -85,B 0,C 180,E1 -3579.628,E2 -3579.628} C_VEL
LIN {X 0,Y 545.079,Z 159.59,A -85,B 0,C 180,E1 -3582.749,E2 -3582.749} C_VEL
LIN {X 0,Y 545.096,Z 159.585,A -85,B 0,C 180,E1 -3585.82,E2 -3585.82} C_VEL
LIN {X 0,Y 545.118,Z 159.58,A -85,B 0,C 180,E1 -3588.849,E2 -3588.849} C_VEL
LIN {X 0,Y 545.066,Z 159.589,A -85,B 0,C 180,E1 -3591.846,E2 -3591.846} C_VEL
LIN {X 0,Y 545.19,Z 159.576,A -85,B 0,C 180,E1 -3594.823,E2 -3594.823} C_VEL
LIN {X 0,Y 545.19,Z 159.573,A -85,B 0,C 180,E1 -3597.784,E2 -3597.784} C_VEL
LIN {X 0,Y 545.214,Z 159.569,A -85,B 0,C 180,E1 -3600.739,E2 -3600.739} C_VEL
LIN {X 0,Y 545.17,Z 159.575,A -85,B 0,C 180,E1 -3602.956,E2 -3602.956} C_VEL
LIN {X 0,Y 545.13,Z 159.578,A -85,B 0,C 180,E1 -3605.92,E2 -3605.92} C_VEL
LIN {X 0,Y 545.09,Z 159.587,A -85,B 0,C 180,E1 -3608.901,E2 -3608.901} C_VEL
LIN {X 0,Y 545.136,Z 159.583,A -85,B 0,C 180,E1 -3611.904,E2 -3611.904} C_VEL
LIN {X 0,Y 545.087,Z 159.586,A -85,B 0,C 180,E1 -3614.944,E2 -3614.944} C_VEL
LIN {X 0,Y 545.072,Z 159.587,A -85,B 0,C 180,E1 -3618.026,E2 -3618.026} C_VEL
LIN {X 0,Y 545.092,Z 159.588,A -85,B 0,C 180,E1 -3620.372,E2 -3620.372} C_VEL
LIN {X 0,Y 545.077,Z 159.586,A -85,B 0,C 180,E1 -3623.56,E2 -3623.56} C_VEL
LIN {X 0,Y 545.076,Z 159.589,A -85,B 0,C 180,E1 -3626.001,E2 -3626.001} C_VEL
LIN {X 0,Y 545.09,Z 159.586,A -85,B 0,C 180,E1 -3628.748,E2 -3628.748} C_VEL
LIN {X 0,Y 545.059,Z 159.588,A -85,B 0,C 180,E1 -3631.679,E2 -3631.679} C_VEL
LIN {X 0,Y 545.059,Z 159.591,A -85,B 0,C 180,E1 -3634.565,E2 -3634.565} C_VEL
LIN {X 0,Y 545.011,Z 159.595,A -85,B 0,C 180,E1 -3637.306,E2 -3637.306} C_VEL
LIN {X 0,Y 545.063,Z 159.587,A -85,B 0,C 180,E1 -3640.143,E2 -3640.143} C_VEL
LIN {X 0,Y 545.08,Z 159.589,A -85,B 0,C 180,E1 -3643.107,E2 -3643.107} C_VEL
LIN {X 0,Y 545.051,Z 159.595,A -85,B 0,C 180,E1 -3646.226,E2 -3646.226} C_VEL
LIN {X 0,Y 545.082,Z 159.586,A -85,B 0,C 180,E1 -3648.885,E2 -3648.885} C_VEL
LIN {X 0,Y 545.042,Z 159.595,A -85,B 0,C 180,E1 -3651.865,E2 -3651.865} C_VEL
LIN {X 0,Y 545.118,Z 159.762,A -85,B 0,C 180,E1 -3652.996,E2 -3652.996} C_VEL
LIN {X 0,Y 545.628,Z 164.681,A -85,B 0,C 180,E1 -3655.027,E2 -3655.027} C_VEL
LIN {X 0,Y 545.504,Z 171.412,A -85,B 0,C 180,E1 -3657.679,E2 -3657.679} C_VEL
LIN {X 0,Y 545.37,Z 179.204,A -85,B 0,C 180,E1 -3660.679,E2 -3660.679} C_VEL
LIN {X 0,Y 545.205,Z 186.995,A -85,B 0,C 180,E1 -3663.594,E2 -3663.594} C_VEL
LIN {X 0,Y 545.104,Z 194.787,A -85,B 0,C 180,E1 -3666.442,E2 -3666.442} C_VEL
LIN {X 0,Y 544.984,Z 202.578,A -85,B 0,C 180,E1 -3669.229,E2 -3669.229} C_VEL
LIN {X 0,Y 544.879,Z 210.369,A -85,B 0,C 180,E1 -3671.967,E2 -3671.967} C_VEL
LIN {X 0,Y 544.815,Z 218.161,A -85,B 0,C 180,E1 -3674.666,E2 -3674.666} C_VEL
LIN {X 0,Y 544.743,Z 224.491,A -85,B 0,C 180,E1 -3676.833,E2 -3676.833} C_VEL
LIN {X 0,Y 546.153,Z 234.348,A -85,B 0,C 180,E1 -3677.08,E2 -3677.08} C_VEL
LIN {X 0,Y 545.968,Z 247.765,A -85,B 0,C 180,E1 -3677.501,E2 -3677.501} C_VEL
LIN {X 0,Y 545.756,Z 259.409,A -85,B 0,C 180,E1 -3678.015,E2 -3678.015} C_VEL
LIN {X 0,Y 545.579,Z 269.752,A -85,B 0,C 180,E1 -3678.605,E2 -3678.605} C_VEL
LIN {X 0,Y 545.406,Z 281.096,A -85,B 0,C 180,E1 -3679.419,E2 -3679.419} C_VEL
LIN {X 0,Y 545.164,Z 291.537,A -85,B 0,C 180,E1 -3680.352,E2 -3680.352} C_VEL
LIN {X 0,Y 545.029,Z 299.989,A -85,B 0,C 180,E1 -3681.285,E2 -3681.285} C_VEL
LIN {X 0,Y 544.86,Z 308.237,A -85,B 0,C 180,E1 -3682.402,E2 -3682.402} C_VEL
LIN {X 0,Y 544.734,Z 315.615,A -85,B 0,C 180,E1 -3683.655,E2 -3683.655} C_VEL
LIN {X 0,Y 544.653,Z 320.949,A -85,B 0,C 180,E1 -3684.818,E2 -3684.818} C_VEL
LIN {X 0,Y 544.684,Z 324.895,A -85,B 0,C 180,E1 -3685.93,E2 -3685.93} C_VEL
LIN {X 0,Y 544.65,Z 327.808,A -85,B 0,C 180,E1 -3687.041,E2 -3687.041} C_VEL
LIN {X 0,Y 544.546,Z 330.185,A -85,B 0,C 180,E1 -3688.521,E2 -3688.521} C_VEL
LIN {X 0,Y 544.541,Z 331,A -85,B 0,C 180,E1 -3690,E2 -3690} C_VEL
LIN {X 0,Y 544.546,Z 330.186,A -85,B 0,C 180,E1 -3691.479,E2 -3691.479} C_VEL
LIN {X 0,Y 544.65,Z 327.81,A -85,B 0,C 180,E1 -3692.958,E2 -3692.958} C_VEL
LIN {X 0,Y 544.684,Z 324.896,A -85,B 0,C 180,E1 -3694.069,E2 -3694.069} C_VEL
LIN {X 0,Y 544.653,Z 320.95,A -85,B 0,C 180,E1 -3695.182,E2 -3695.182} C_VEL
LIN {X 0,Y 544.737,Z 315.595,A -85,B 0,C 180,E1 -3696.349,E2 -3696.349} C_VEL
LIN {X 0,Y 544.859,Z 308.239,A -85,B 0,C 180,E1 -3697.597,E2 -3697.597} C_VEL
LIN {X 0,Y 545.029,Z 299.992,A -85,B 0,C 180,E1 -3698.714,E2 -3698.714} C_VEL
LIN {X 0,Y 545.162,Z 291.54,A -85,B 0,C 180,E1 -3699.648,E2 -3699.648} C_VEL
LIN {X 0,Y 545.406,Z 281.1,A -85,B 0,C 180,E1 -3700.581,E2 -3700.581} C_VEL
LIN {X 0,Y 545.587,Z 269.668,A -85,B 0,C 180,E1 -3701.401,E2 -3701.401} C_VEL
LIN {X 0,Y 545.761,Z 259.415,A -85,B 0,C 180,E1 -3701.984,E2 -3701.984} C_VEL
LIN {X 0,Y 545.966,Z 247.77,A -85,B 0,C 180,E1 -3702.499,E2 -3702.499} C_VEL
LIN {X 0,Y 546.153,Z 234.358,A -85,B 0,C 180,E1 -3702.919,E2 -3702.919} C_VEL
LIN {X 0,Y 544.744,Z 224.492,A -85,B 0,C 180,E1 -3703.167,E2 -3703.167} C_VEL
LIN {X 0,Y 544.84,Z 217.049,A -85,B 0,C 180,E1 -3705.717,E2 -3705.717} C_VEL
LIN {X 0,Y 544.906,Z 208.144,A -85,B 0,C 180,E1 -3708.81,E2 -3708.81} C_VEL
LIN {X 0,Y 544.999,Z 201.466,A -85,B 0,C 180,E1 -3711.166,E2 -3711.166} C_VEL
LIN {X 0,Y 545.143,Z 192.562,A -85,B 0,C 180,E1 -3714.364,E2 -3714.364} C_VEL
LIN {X 0,Y 545.283,Z 184.817,A -85,B 0,C 180,E1 -3717.211,E2 -3717.211} C_VEL
LIN {X 0,Y 545.406,Z 176.623,A -85,B 0,C 180,E1 -3720.305,E2 -3720.305} C_VEL
LIN {X 0,Y 545.522,Z 169.341,A -85,B 0,C 180,E1 -3723.133,E2 -3723.133} C_VEL
LIN {X 0,Y 545.6,Z 163.558,A -85,B 0,C 180,E1 -3725.426,E2 -3725.426} C_VEL
LIN {X 0,Y 545.073,Z 159.592,A -85,B 0,C 180,E1 -3727.135,E2 -3727.135} C_VEL
LIN {X 0,Y 545.062,Z 159.594,A -85,B 0,C 180,E1 -3730.143,E2 -3730.143} C_VEL
LIN {X 0,Y 545.079,Z 159.586,A -85,B 0,C 180,E1 -3733.106,E2 -3733.106} C_VEL
LIN {X 0,Y 545.048,Z 159.589,A -85,B 0,C 180,E1 -3736.226,E2 -3736.226} C_VEL
LIN {X 0,Y 545.08,Z 159.591,A -85,B 0,C 180,E1 -3738.885,E2 -3738.885} C_VEL
LIN {X 0,Y 545.074,Z 159.589,A -85,B 0,C 180,E1 -3740.818,E2 -3740.818} C_VEL
LIN {X 0,Y 545.012,Z 159.596,A -85,B 0,C 180,E1 -3743.617,E2 -3743.617} C_VEL
LIN {X 0,Y 545.063,Z 159.588,A -85,B 0,C 180,E1 -3746.328,E2 -3746.328} C_VEL
LIN {X 0,Y 545.066,Z 159.592,A -85,B 0,C 180,E1 -3748.952,E2 -3748.952} C_VEL
LIN {X 0,Y 545.101,Z 159.583,A -85,B 0,C 180,E1 -3751.508,E2 -3751.508} C_VEL
LIN {X 0,Y 545.093,Z 159.587,A -85,B 0,C 180,E1 -3754.491,E2 -3754.491} C_VEL
LIN {X 0,Y 545.03,Z 159.592,A -85,B 0,C 180,E1 -3757.242,E2 -3757.242} C_VEL
LIN {X 0,Y 545.114,Z 159.581,A -85,B 0,C 180,E1 -3760.415,E2 -3760.415} C_VEL
LIN {X 0,Y 545.072,Z 159.587,A -85,B 0,C 180,E1 -3763.521,E2 -3763.521} C_VEL
LIN {X 0,Y 545.093,Z 159.586,A -85,B 0,C 180,E1 -3765.82,E2 -3765.82} C_VEL
LIN {X 0,Y 545.114,Z 159.581,A -85,B 0,C 180,E1 -3768.849,E2 -3768.849} C_VEL
LIN {X 0,Y 545.063,Z 159.588,A -85,B 0,C 180,E1 -3771.846,E2 -3771.846} C_VEL
LIN {X 0,Y 545.192,Z 159.577,A -85,B 0,C 180,E1 -3774.823,E2 -3774.823} C_VEL
LIN {X 0,Y 545.191,Z 159.573,A -85,B 0,C 180,E1 -3777.784,E2 -3777.784} C_VEL
LIN {X 0,Y 545.212,Z 159.569,A -85,B 0,C 180,E1 -3780.739,E2 -3780.739} C_VEL
LIN {X 0,Y 545.168,Z 159.576,A -85,B 0,C 180,E1 -3782.956,E2 -3782.956} C_VEL
LIN {X 0,Y 545.126,Z 159.579,A -85,B 0,C 180,E1 -3785.92,E2 -3785.92} C_VEL
LIN {X 0,Y 545.091,Z 159.585,A -85,B 0,C 180,E1 -3788.901,E2 -3788.901} C_VEL
LIN {X 0,Y 545.133,Z 159.583,A -85,B 0,C 180,E1 -3791.904,E2 -3791.904} C_VEL
LIN {X 0,Y 545.084,Z 159.587,A -85,B 0,C 180,E1 -3794.944,E2 -3794.944} C_VEL
LIN {X 0,Y 545.075,Z 159.586,A -85,B 0,C 180,E1 -3798.026,E2 -3798.026} C_VEL
LIN {X 0,Y 545.089,Z 159.589,A -85,B 0,C 180,E1 -3800.372,E2 -3800.372} C_VEL
LIN {X 0,Y 545.074,Z 159.587,A -85,B 0,C 180,E1 -3803.56,E2 -3803.56} C_VEL
LIN {X 0,Y 545.078,Z 159.588,A -85,B 0,C 180,E1 -3806.001,E2 -3806.001} C_VEL
LIN {X 0,Y 545.088,Z 159.587,A -85,B 0,C 180,E1 -3808.748,E2 -3808.748} C_VEL
LIN {X 0,Y 545.056,Z 159.589,A -85,B 0,C 180,E1 -3811.679,E2 -3811.679} C_VEL
LIN {X 0,Y 545.057,Z 159.592,A -85,B 0,C 180,E1 -3814.565,E2 -3814.565} C_VEL
LIN {X 0,Y 545.012,Z 159.594,A -85,B 0,C 180,E1 -3816.993,E2 -3816.993} C_VEL
LIN {X 0,Y 544.346,Z 159.683,A -85,B 0,C 180,E1 -3817.609,E2 -3817.609} C_VEL
LIN {X 0,Y 541.501,Z 160.033,A -85,B 0,C 180,E1 -3818.611,E2 -3818.611} C_VEL
LIN {X 0,Y 539.106,Z 160.335,A -85,B 0,C 180,E1 -3819.417,E2 -3819.417} C_VEL
LIN {X 0,Y 538.09,Z 160.456,A -85,B 0,C 180,E1 -3820.04,E2 -3820.04} C_VEL
LIN {X 0,Y 538.014,Z 160.465,A -85,B 0,C 180,E1 -3820.25,E2 -3820.25} C_VEL
LIN {X 0,Y 538.026,Z 160.469,A -85,B 0,C 180,E1 -3822.988,E2 -3822.988} C_VEL
LIN {X 0,Y 538.024,Z 160.467,A -85,B 0,C 180,E1 -3825.926,E2 -3825.926} C_VEL
LIN {X 0,Y 538.048,Z 160.464,A -85,B 0,C 180,E1 -3829.225,E2 -3829.225} C_VEL
LIN {X 0,Y 537.982,Z 160.47,A -85,B 0,C 180,E1 -3832.122,E2 -3832.122} C_VEL
LIN {X 0,Y 537.941,Z 160.476,A -85,B 0,C 180,E1 -3834.097,E2 -3834.097} C_VEL
LIN {X 0,Y 537.902,Z 160.889,A -85,B 0,C 180,E1 -3834.909,E2 -3834.909} C_VEL
LIN {X 0,Y 537.882,Z 165.079,A -85,B 0,C 180,E1 -3837.608,E2 -3837.608} C_VEL
LIN {X 0,Y 537.87,Z 169.2,A -85,B 0,C 180,E1 -3840.23,E2 -3840.23} C_VEL
LIN {X 0,Y 537.813,Z 173.287,A -85,B 0,C 180,E1 -3842.783,E2 -3842.783} C_VEL
LIN {X 0,Y 537.791,Z 177.358,A -85,B 0,C 180,E1 -3845.28,E2 -3845.28} C_VEL
LIN {X 0,Y 537.73,Z 182.797,A -85,B 0,C 180,E1 -3848.534,E2 -3848.534} C_VEL
LIN {X 0,Y 537.652,Z 186.872,A -85,B 0,C 180,E1 -3850.926,E2 -3850.926} C_VEL
LIN {X 0,Y 537.595,Z 190.954,A -85,B 0,C 180,E1 -3853.286,E2 -3853.286} C_VEL
LIN {X 0,Y 537.574,Z 195.059,A -85,B 0,C 180,E1 -3855.618,E2 -3855.618} C_VEL
LIN {X 0,Y 537.55,Z 197.018,A -85,B 0,C 180,E1 -3856.738,E2 -3856.738} C_VEL
LIN {X 0,Y 539.212,Z 206.722,A -85,B 0,C 180,E1 -3857.007,E2 -3857.007} C_VEL
LIN {X 0,Y 539.033,Z 219.453,A -85,B 0,C 180,E1 -3857.434,E2 -3857.434} C_VEL
LIN {X 0,Y 538.779,Z 232.029,A -85,B 0,C 180,E1 -3858.024,E2 -3858.024} C_VEL
LIN {X 0,Y 538.558,Z 243.279,A -85,B 0,C 180,E1 -3858.712,E2 -3858.712} C_VEL
LIN {X 0,Y 538.335,Z 254.275,A -85,B 0,C 180,E1 -3859.564,E2 -3859.564} C_VEL
LIN {X 0,Y 538.108,Z 264.963,A -85,B 0,C 180,E1 -3860.604,E2 -3860.604} C_VEL
LIN {X 0,Y 537.954,Z 272.844,A -85,B 0,C 180,E1 -3861.549,E2 -3861.549} C_VEL
LIN {X 0,Y 537.788,Z 280.552,A -85,B 0,C 180,E1 -3862.68,E2 -3862.68} C_VEL
LIN {X 0,Y 537.717,Z 287.618,A -85,B 0,C 180,E1 -3863.998,E2 -3863.998} C_VEL
LIN {X 0,Y 537.54,Z 292.332,A -85,B 0,C 180,E1 -3865.125,E2 -3865.125} C_VEL
LIN {X 0,Y 537.591,Z 295.938,A -85,B 0,C 180,E1 -3866.252,E2 -3866.252} C_VEL
LIN {X 0,Y 537.58,Z 297.803,A -85,B 0,C 180,E1 -3867.003,E2 -3867.003} C_VEL
LIN {X 0,Y 537.49,Z 299.214,A -85,B 0,C 180,E1 -3867.752,E2 -3867.752} C_VEL
LIN {X 0,Y 537.443,Z 300.833,A -85,B 0,C 180,E1 -3869.251,E2 -3869.251} C_VEL
LIN {X 0,Y 537.443,Z 301.071,A -85,B 0,C 180,E1 -3870,E2 -3870} C_VEL
LIN {X 0,Y 537.442,Z 300.889,A -85,B 0,C 180,E1 -3870.749,E2 -3870.749} C_VEL
LIN {X 0,Y 537.49,Z 299.344,A -85,B 0,C 180,E1 -3872.248,E2 -3872.248} C_VEL
LIN {X 0,Y 537.58,Z 297.99,A -85,B 0,C 180,E1 -3872.998,E2 -3872.998} C_VEL
LIN {X 0,Y 537.604,Z 295.131,A -85,B 0,C 180,E1 -3874.123,E2 -3874.123} C_VEL
LIN {X 0,Y 537.587,Z 291.255,A -85,B 0,C 180,E1 -3875.251,E2 -3875.251} C_VEL
LIN {X 0,Y 537.662,Z 286.529,A -85,B 0,C 180,E1 -3876.321,E2 -3876.321} C_VEL
LIN {X 0,Y 537.79,Z 279.954,A -85,B 0,C 180,E1 -3877.509,E2 -3877.509} C_VEL
LIN {X 0,Y 537.961,Z 272.067,A -85,B 0,C 180,E1 -3878.641,E2 -3878.641} C_VEL
LIN {X 0,Y 538.182,Z 262.253,A -85,B 0,C 180,E1 -3879.774,E2 -3879.774} C_VEL
LIN {X 0,Y 538.387,Z 251.965,A -85,B 0,C 180,E1 -3880.721,E2 -3880.721} C_VEL
LIN {X 0,Y 538.58,Z 241.217,A -85,B 0,C 180,E1 -3881.516,E2 -3881.516} C_VEL
LIN {X 0,Y 538.82,Z 230.62,A -85,B 0,C 180,E1 -3882.141,E2 -3882.141} C_VEL
LIN {X 0,Y 539.064,Z 218.105,A -85,B 0,C 180,E1 -3882.71,E2 -3882.71} C_VEL
LIN {X 0,Y 539.045,Z 205.243,A -85,B 0,C 180,E1 -3883.126,E2 -3883.126} C_VEL
LIN {X 0,Y 537.544,Z 196.924,A -85,B 0,C 180,E1 -3883.371,E2 -3883.371} C_VEL
LIN {X 0,Y 537.575,Z 192.473,A -85,B 0,C 180,E1 -3885.935,E2 -3885.935} C_VEL
LIN {X 0,Y 537.607,Z 188.38,A -85,B 0,C 180,E1 -3888.285,E2 -3888.285} C_VEL
LIN {X 0,Y 537.668,Z 184.308,A -85,B 0,C 180,E1 -3890.666,E2 -3890.666} C_VEL
LIN {X 0,Y 537.716,Z 180.231,A -85,B 0,C 180,E1 -3893.086,E2 -3893.086} C_VEL
LIN {X 0,Y 537.788,Z 176.039,A -85,B 0,C 180,E1 -3895.615,E2 -3895.615} C_VEL
LIN {X 0,Y 537.826,Z 172.074,A -85,B 0,C 180,E1 -3898.062,E2 -3898.062} C_VEL
LIN {X 0,Y 537.891,Z 167.982,A -85,B 0,C 180,E1 -3900.635,E2 -3900.635} C_VEL
LIN {X 0,Y 537.953,Z 163.838,A -85,B 0,C 180,E1 -3903.278,E2 -3903.278} C_VEL
LIN {X 0,Y 537.949,Z 161.028,A -85,B 0,C 180,E1 -3905.088,E2 -3905.088} C_VEL
LIN {X 0,Y 537.954,Z 160.474,A -85,B 0,C 180,E1 -3906.008,E2 -3906.008} C_VEL
LIN {X 0,Y 537.989,Z 160.474,A -85,B 0,C 180,E1 -3908.833,E2 -3908.833} C_VEL
LIN {X 0,Y 538.002,Z 160.471,A -85,B 0,C 180,E1 -3911.875,E2 -3911.875} C_VEL
LIN {X 0,Y 538.009,Z 160.467,A -85,B 0,C 180,E1 -3914.862,E2 -3914.862} C_VEL
LIN {X 0,Y 538.021,Z 160.471,A -85,B 0,C 180,E1 -3917.214,E2 -3917.214} C_VEL
LIN {X 0,Y 538.022,Z 160.465,A -85,B 0,C 180,E1 -3920.203,E2 -3920.203} C_VEL
LIN {X 0,Y 537.971,Z 160.471,A -85,B 0,C 180,E1 -3923.063,E2 -3923.063} C_VEL
LIN {X 0,Y 538.001,Z 160.472,A -85,B 0,C 180,E1 -3925.825,E2 -3925.825} C_VEL
LIN {X 0,Y 538.01,Z 160.467,A -85,B 0,C 180,E1 -3928.499,E2 -3928.499} C_VEL
LIN {X 0,Y 538.062,Z 160.463,A -85,B 0,C 180,E1 -3931.1,E2 -3931.1} C_VEL
LIN {X 0,Y 538.043,Z 160.461,A -85,B 0,C 180,E1 -3933.633,E2 -3933.633} C_VEL
LIN {X 0,Y 538.008,Z 160.473,A -85,B 0,C 180,E1 -3936.122,E2 -3936.122} C_VEL
LIN {X 0,Y 538.037,Z 160.466,A -85,B 0,C 180,E1 -3939.348,E2 -3939.348} C_VEL
LIN {X 0,Y 538.037,Z 160.465,A -85,B 0,C 180,E1 -3942.468,E2 -3942.468} C_VEL
LIN {X 0,Y 538.065,Z 160.46,A -85,B 0,C 180,E1 -3945.631,E2 -3945.631} C_VEL
LIN {X 0,Y 538.078,Z 160.458,A -85,B 0,C 180,E1 -3948.701,E2 -3948.701} C_VEL
LIN {X 0,Y 538.038,Z 160.466,A -85,B 0,C 180,E1 -3951.739,E2 -3951.739} C_VEL
LIN {X 0,Y 538.145,Z 160.453,A -85,B 0,C 180,E1 -3954.755,E2 -3954.755} C_VEL
LIN {X 0,Y 538.163,Z 160.448,A -85,B 0,C 180,E1 -3957.755,E2 -3957.755} C_VEL
LIN {X 0,Y 538.184,Z 160.445,A -85,B 0,C 180,E1 -3960.748,E2 -3960.748} C_VEL
LIN {X 0,Y 538.137,Z 160.452,A -85,B 0,C 180,E1 -3962.994,E2 -3962.994} C_VEL
LIN {X 0,Y 538.087,Z 160.456,A -85,B 0,C 180,E1 -3965.998,E2 -3965.998} C_VEL
LIN {X 0,Y 538.044,Z 160.464,A -85,B 0,C 180,E1 -3969.018,E2 -3969.018} C_VEL
LIN {X 0,Y 538.084,Z 160.462,A -85,B 0,C 180,E1 -3972.063,E2 -3972.063} C_VEL
LIN {X 0,Y 538.047,Z 160.465,A -85,B 0,C 180,E1 -3975.144,E2 -3975.144} C_VEL
LIN {X 0,Y 538.026,Z 160.465,A -85,B 0,C 180,E1 -3978.27,E2 -3978.27} C_VEL
LIN {X 0,Y 538.037,Z 160.468,A -85,B 0,C 180,E1 -3980.651,E2 -3980.651} C_VEL
LIN {X 0,Y 538.001,Z 160.471,A -85,B 0,C 180,E1 -3983.889,E2 -3983.889} C_VEL
LIN {X 0,Y 538.038,Z 160.463,A -85,B 0,C 180,E1 -3986.367,E2 -3986.367} C_VEL
LIN {X 0,Y 538.032,Z 160.468,A -85,B 0,C 180,E1 -3988.933,E2 -3988.933} C_VEL
LIN {X 0,Y 538.012,Z 160.467,A -85,B 0,C 180,E1 -3991.887,E2 -3991.887} C_VEL
LIN {X 0,Y 538.008,Z 160.469,A -85,B 0,C 180,E1 -3994.617,E2 -3994.617} C_VEL
LIN {X 0,Y 537.979,Z 160.474,A -85,B 0,C 180,E1 -3997.879,E2 -3997.879} C_VEL
LIN {X 0,Y 538.049,Z 160.463,A -85,B 0,C 180,E1 -4000.776,E2 -4000.776} C_VEL
LIN {X 0,Y 538.005,Z 160.467,A -85,B 0,C 180,E1 -4003.816,E2 -4003.816} C_VEL
LIN {X 0,Y 538.028,Z 160.464,A -85,B 0,C 180,E1 -4007.013,E2 -4007.013} C_VEL
LIN {X 0,Y 538.049,Z 160.463,A -85,B 0,C 180,E1 -4009.253,E2 -4009.253} C_VEL
LIN {X 0,Y 538.032,Z 160.468,A -85,B 0,C 180,E1 -4012.509,E2 -4012.509} C_VEL
LIN {X 0,Y 538.059,Z 160.638,A -85,B 0,C 180,E1 -4012.823,E2 -4012.823} C_VEL
LIN {X 0,Y 538.594,Z 164.618,A -85,B 0,C 180,E1 -4014.502,E2 -4014.502} C_VEL
LIN {X 0,Y 538.492,Z 171.367,A -85,B 0,C 180,E1 -4017.205,E2 -4017.205} C_VEL
LIN {X 0,Y 538.39,Z 177.22,A -85,B 0,C 180,E1 -4019.491,E2 -4019.491} C_VEL
LIN {X 0,Y 538.264,Z 185.351,A -85,B 0,C 180,E1 -4022.606,E2 -4022.606} C_VEL
LIN {X 0,Y 538.1,Z 193.675,A -85,B 0,C 180,E1 -4025.707,E2 -4025.707} C_VEL
LIN {X 0,Y 537.98,Z 201.465,A -85,B 0,C 180,E1 -4028.544,E2 -4028.544} C_VEL
LIN {X 0,Y 537.846,Z 209.256,A -85,B 0,C 180,E1 -4031.328,E2 -4031.328} C_VEL
LIN {X 0,Y 537.758,Z 217.048,A -85,B 0,C 180,E1 -4034.071,E2 -4034.071} C_VEL
LIN {X 0,Y 537.69,Z 224.491,A -85,B 0,C 180,E1 -4036.657,E2 -4036.657} C_VEL
LIN {X 0,Y 539.241,Z 234.348,A -85,B 0,C 180,E1 -4036.912,E2 -4036.912} C_VEL
LIN {X 0,Y 539.034,Z 247.765,A -85,B 0,C 180,E1 -4037.338,E2 -4037.338} C_VEL
LIN {X 0,Y 538.816,Z 259.409,A -85,B 0,C 180,E1 -4037.858,E2 -4037.858} C_VEL
LIN {X 0,Y 538.603,Z 270.162,A -85,B 0,C 180,E1 -4038.482,E2 -4038.482} C_VEL
LIN {X 0,Y 538.372,Z 281.097,A -85,B 0,C 180,E1 -4039.279,E2 -4039.279} C_VEL
LIN {X 0,Y 538.137,Z 291.537,A -85,B 0,C 180,E1 -4040.225,E2 -4040.225} C_VEL
LIN {X 0,Y 537.974,Z 299.989,A -85,B 0,C 180,E1 -4041.17,E2 -4041.17} C_VEL
LIN {X 0,Y 537.817,Z 308.237,A -85,B 0,C 180,E1 -4042.302,E2 -4042.302} C_VEL
LIN {X 0,Y 537.683,Z 314.75,A -85,B 0,C 180,E1 -4043.409,E2 -4043.409} C_VEL
LIN {X 0,Y 537.676,Z 319.365,A -85,B 0,C 180,E1 -4044.374,E2 -4044.374} C_VEL
LIN {X 0,Y 537.557,Z 323.677,A -85,B 0,C 180,E1 -4045.501,E2 -4045.501} C_VEL
LIN {X 0,Y 537.591,Z 325.957,A -85,B 0,C 180,E1 -4046.252,E2 -4046.252} C_VEL
LIN {X 0,Y 537.551,Z 327.808,A -85,B 0,C 180,E1 -4047.002,E2 -4047.002} C_VEL
LIN {X 0,Y 537.49,Z 329.198,A -85,B 0,C 180,E1 -4047.752,E2 -4047.752} C_VEL
LIN {X 0,Y 537.442,Z 330.785,A -85,B 0,C 180,E1 -4049.251,E2 -4049.251} C_VEL
LIN {X 0,Y 537.442,Z 331,A -85,B 0,C 180,E1 -4050,E2 -4050} C_VEL
LIN {X 0,Y 537.451,Z 330.187,A -85,B 0,C 180,E1 -4051.498,E2 -4051.498} C_VEL
LIN {X 0,Y 537.49,Z 329.2,A -85,B 0,C 180,E1 -4052.248,E2 -4052.248} C_VEL
LIN {X 0,Y 537.551,Z 327.81,A -85,B 0,C 180,E1 -4052.998,E2 -4052.998} C_VEL
LIN {X 0,Y 537.603,Z 324.896,A -85,B 0,C 180,E1 -4054.123,E2 -4054.123} C_VEL
LIN {X 0,Y 537.587,Z 320.95,A -85,B 0,C 180,E1 -4055.25,E2 -4055.25} C_VEL
LIN {X 0,Y 537.652,Z 316.087,A -85,B 0,C 180,E1 -4056.334,E2 -4056.334} C_VEL
LIN {X 0,Y 537.79,Z 309.47,A -85,B 0,C 180,E1 -4057.509,E2 -4057.509} C_VEL
LIN {X 0,Y 537.972,Z 301.48,A -85,B 0,C 180,E1 -4058.64,E2 -4058.64} C_VEL
LIN {X 0,Y 538.117,Z 293.338,A -85,B 0,C 180,E1 -4059.585,E2 -4059.585} C_VEL
LIN {X 0,Y 538.363,Z 283.404,A -85,B 0,C 180,E1 -4060.53,E2 -4060.53} C_VEL
LIN {X 0,Y 538.531,Z 273.59,A -85,B 0,C 180,E1 -4061.289,E2 -4061.289} C_VEL
LIN {X 0,Y 538.715,Z 262.593,A -85,B 0,C 180,E1 -4061.971,E2 -4061.971} C_VEL
LIN {X 0,Y 538.968,Z 250.116,A -85,B 0,C 180,E1 -4062.568,E2 -4062.568} C_VEL
LIN {X 0,Y 539.194,Z 237.099,A -85,B 0,C 180,E1 -4063.017,E2 -4063.017} C_VEL
LIN {X 0,Y 538.964,Z 232.173,A -85,B 0,C 180,E1 -4063.152,E2 -4063.152} C_VEL
LIN {X 0,Y 537.69,Z 224.492,A -85,B 0,C 180,E1 -4063.343,E2 -4063.343} C_VEL
LIN {X 0,Y 537.757,Z 217.049,A -85,B 0,C 180,E1 -4065.929,E2 -4065.929} C_VEL
LIN {X 0,Y 537.845,Z 209.257,A -85,B 0,C 180,E1 -4068.671,E2 -4068.671} C_VEL
LIN {X 0,Y 537.982,Z 201.466,A -85,B 0,C 180,E1 -4071.455,E2 -4071.455} C_VEL
LIN {X 0,Y 538.099,Z 193.676,A -85,B 0,C 180,E1 -4074.293,E2 -4074.293} C_VEL
LIN {X 0,Y 538.263,Z 185.352,A -85,B 0,C 180,E1 -4077.394,E2 -4077.394} C_VEL
LIN {X 0,Y 538.409,Z 176.979,A -85,B 0,C 180,E1 -4080.602,E2 -4080.602} C_VEL
LIN {X 0,Y 538.536,Z 169.925,A -85,B 0,C 180,E1 -4083.362,E2 -4083.362} C_VEL
LIN {X 0,Y 538.601,Z 164.608,A -85,B 0,C 180,E1 -4085.497,E2 -4085.497} C_VEL
LIN {X 0,Y 538.039,Z 160.468,A -85,B 0,C 180,E1 -4087.3,E2 -4087.3} C_VEL
LIN {X 0,Y 538.007,Z 160.47,A -85,B 0,C 180,E1 -4089.798,E2 -4089.798} C_VEL
LIN {X 0,Y 538.019,Z 160.466,A -85,B 0,C 180,E1 -4092.786,E2 -4092.786} C_VEL
LIN {X 0,Y 538.018,Z 160.467,A -85,B 0,C 180,E1 -4095.926,E2 -4095.926} C_VEL
LIN {X 0,Y 538.029,Z 160.464,A -85,B 0,C 180,E1 -4098.226,E2 -4098.226} C_VEL
LIN {X 0,Y 538.006,Z 160.466,A -85,B 0,C 180,E1 -4101.169,E2 -4101.169} C_VEL
LIN {X 0,Y 537.963,Z 160.478,A -85,B 0,C 180,E1 -4104.093,E2 -4104.093} C_VEL
LIN {X 0,Y 538.029,Z 160.464,A -85,B 0,C 180,E1 -4106.727,E2 -4106.727} C_VEL
LIN {X 0,Y 538.025,Z 160.467,A -85,B 0,C 180,E1 -4109.556,E2 -4109.556} C_VEL
LIN {X 0,Y 538.043,Z 160.463,A -85,B 0,C 180,E1 -4111.95,E2 -4111.95} C_VEL
LIN {X 0,Y 538.069,Z 160.462,A -85,B 0,C 180,E1 -4114.467,E2 -4114.467} C_VEL
LIN {X 0,Y 537.989,Z 160.475,A -85,B 0,C 180,E1 -4117.738,E2 -4117.738} C_VEL
LIN {X 0,Y 538.078,Z 160.458,A -85,B 0,C 180,E1 -4120.148,E2 -4120.148} C_VEL
LIN {X 0,Y 538.023,Z 160.467,A -85,B 0,C 180,E1 -4123.299,E2 -4123.299} C_VEL
LIN {X 0,Y 538.062,Z 160.461,A -85,B 0,C 180,E1 -4125.631,E2 -4125.631} C_VEL
LIN {X 0,Y 538.074,Z 160.458,A -85,B 0,C 180,E1 -4128.701,E2 -4128.701} C_VEL
LIN {X 0,Y 538.035,Z 160.465,A -85,B 0,C 180,E1 -4131.739,E2 -4131.739} C_VEL
LIN {X 0,Y 538.147,Z 160.453,A -85,B 0,C 180,E1 -4134.755,E2 -4134.755} C_VEL
LIN {X 0,Y 538.163,Z 160.448,A -85,B 0,C 180,E1 -4137.755,E2 -4137.755} C_VEL
LIN {X 0,Y 538.182,Z 160.445,A -85,B 0,C 180,E1 -4140.748,E2 -4140.748} C_VEL
LIN {X 0,Y 538.135,Z 160.453,A -85,B 0,C 180,E1 -4142.995,E2 -4142.995} C_VEL
LIN {X 0,Y 538.083,Z 160.457,A -85,B 0,C 180,E1 -4145.998,E2 -4145.998} C_VEL
LIN {X 0,Y 538.045,Z 160.462,A -85,B 0,C 180,E1 -4149.018,E2 -4149.018} C_VEL
LIN {X 0,Y 538.081,Z 160.463,A -85,B 0,C 180,E1 -4152.063,E2 -4152.063} C_VEL
LIN {X 0,Y 538.044,Z 160.466,A -85,B 0,C 180,E1 -4155.144,E2 -4155.144} C_VEL
LIN {X 0,Y 538.027,Z 160.465,A -85,B 0,C 180,E1 -4158.27,E2 -4158.27} C_VEL
LIN {X 0,Y 538.034,Z 160.467,A -85,B 0,C 180,E1 -4160.652,E2 -4160.652} C_VEL
LIN {X 0,Y 537.999,Z 160.473,A -85,B 0,C 180,E1 -4163.889,E2 -4163.889} C_VEL
LIN {X 0,Y 538.04,Z 160.462,A -85,B 0,C 180,E1 -4166.367,E2 -4166.367} C_VEL
LIN {X 0,Y 538.029,Z 160.467,A -85,B 0,C 180,E1 -4168.934,E2 -4168.934} C_VEL
LIN {X 0,Y 538.009,Z 160.467,A -85,B 0,C 180,E1 -4171.888,E2 -4171.888} C_VEL
LIN {X 0,Y 538.006,Z 160.469,A -85,B 0,C 180,E1 -4174.617,E2 -4174.617} C_VEL
LIN {X 0,Y 537.98,Z 160.473,A -85,B 0,C 180,E1 -4177.879,E2 -4177.879} C_VEL
LIN {X 0,Y 538.014,Z 160.465,A -85,B 0,C 180,E1 -4180.25,E2 -4180.25} C_VEL
LIN {X 0,Y 537.365,Z 160.551,A -85,B 0,C 180,E1 -4180.876,E2 -4180.876} C_VEL
LIN {X 0,Y 534.512,Z 160.904,A -85,B 0,C 180,E1 -4181.89,E2 -4181.89} C_VEL
LIN {X 0,Y 532.087,Z 161.208,A -85,B 0,C 180,E1 -4182.708,E2 -4182.708} C_VEL
LIN {X 0,Y 531.04,Z 161.336,A -85,B 0,C 180,E1 -4183.339,E2 -4183.339} C_VEL
LIN {X 0,Y 530.952,Z 161.345,A -85,B 0,C 180,E1 -4183.552,E2 -4183.552} C_VEL
LIN {X 0,Y 530.959,Z 161.349,A -85,B 0,C 180,E1 -4186.505,E2 -4186.505} C_VEL
LIN {X 0,Y 530.983,Z 161.342,A -85,B 0,C 180,E1 -4188.977,E2 -4188.977} C_VEL
LIN {X 0,Y 530.948,Z 161.35,A -85,B 0,C 180,E1 -4191.529,E2 -4191.529} C_VEL
LIN {X 0,Y 530.87,Z 161.358,A -85,B 0,C 180,E1 -4194.374,E2 -4194.374} C_VEL
LIN {X 0,Y 530.901,Z 162.366,A -85,B 0,C 180,E1 -4195.304,E2 -4195.304} C_VEL
LIN {X 0,Y 530.845,Z 166.54,A -85,B 0,C 180,E1 -4198.024,E2 -4198.024} C_VEL
LIN {X 0,Y 530.805,Z 171.048,A -85,B 0,C 180,E1 -4200.911,E2 -4200.911} C_VEL
LIN {X 0,Y 530.728,Z 176.119,A -85,B 0,C 180,E1 -4204.088,E2 -4204.088} C_VEL
LIN {X 0,Y 530.678,Z 180.191,A -85,B 0,C 180,E1 -4206.591,E2 -4206.591} C_VEL
LIN {X 0,Y 530.619,Z 184.279,A -85,B 0,C 180,E1 -4209.047,E2 -4209.047} C_VEL
LIN {X 0,Y 530.54,Z 188.374,A -85,B 0,C 180,E1 -4211.463,E2 -4211.463} C_VEL
LIN {X 0,Y 530.494,Z 192.478,A -85,B 0,C 180,E1 -4213.847,E2 -4213.847} C_VEL
LIN {X 0,Y 530.492,Z 197.216,A -85,B 0,C 180,E1 -4216.546,E2 -4216.546} C_VEL
LIN {X 0,Y 532.332,Z 207.865,A -85,B 0,C 180,E1 -4216.86,E2 -4216.86} C_VEL
LIN {X 0,Y 532.074,Z 220.808,A -85,B 0,C 180,E1 -4217.315,E2 -4217.315} C_VEL
LIN {X 0,Y 531.828,Z 232.41,A -85,B 0,C 180,E1 -4217.874,E2 -4217.874} C_VEL
LIN {X 0,Y 531.594,Z 243.501,A -85,B 0,C 180,E1 -4218.562,E2 -4218.562} C_VEL
LIN {X 0,Y 531.349,Z 254.495,A -85,B 0,C 180,E1 -4219.425,E2 -4219.425} C_VEL
LIN {X 0,Y 531.103,Z 265.182,A -85,B 0,C 180,E1 -4220.479,E2 -4220.479} C_VEL
LIN {X 0,Y 530.942,Z 273.061,A -85,B 0,C 180,E1 -4221.436,E2 -4221.436} C_VEL
LIN {X 0,Y 530.733,Z 280.769,A -85,B 0,C 180,E1 -4222.582,E2 -4222.582} C_VEL
LIN {X 0,Y 530.652,Z 287.834,A -85,B 0,C 180,E1 -4223.918,E2 -4223.918} C_VEL
LIN {X 0,Y 530.459,Z 292.548,A -85,B 0,C 180,E1 -4225.06,E2 -4225.06} C_VEL
LIN {X 0,Y 530.516,Z 296.152,A -85,B 0,C 180,E1 -4226.202,E2 -4226.202} C_VEL
LIN {X 0,Y 530.512,Z 298.017,A -85,B 0,C 180,E1 -4226.963,E2 -4226.963} C_VEL
LIN {X 0,Y 530.412,Z 299.427,A -85,B 0,C 180,E1 -4227.722,E2 -4227.722} C_VEL
LIN {X 0,Y 530.346,Z 301.046,A -85,B 0,C 180,E1 -4229.241,E2 -4229.241} C_VEL
LIN {X 0,Y 530.347,Z 301.284,A -85,B 0,C 180,E1 -4230,E2 -4230} C_VEL
LIN {X 0,Y 530.346,Z 301.102,A -85,B 0,C 180,E1 -4230.759,E2 -4230.759} C_VEL
LIN {X 0,Y 530.413,Z 299.556,A -85,B 0,C 180,E1 -4232.278,E2 -4232.278} C_VEL
LIN {X 0,Y 530.512,Z 298.201,A -85,B 0,C 180,E1 -4233.038,E2 -4233.038} C_VEL
LIN {X 0,Y 530.523,Z 295.343,A -85,B 0,C 180,E1 -4234.178,E2 -4234.178} C_VEL
LIN {X 0,Y 530.524,Z 291.466,A -85,B 0,C 180,E1 -4235.321,E2 -4235.321} C_VEL
LIN {X 0,Y 530.605,Z 285.854,A -85,B 0,C 180,E1 -4236.587,E2 -4236.587} C_VEL
LIN {X 0,Y 530.793,Z 278.941,A -85,B 0,C 180,E1 -4237.8,E2 -4237.8} C_VEL
LIN {X 0,Y 530.958,Z 270.797,A -85,B 0,C 180,E1 -4238.948,E2 -4238.948} C_VEL
LIN {X 0,Y 531.186,Z 262.461,A -85,B 0,C 180,E1 -4239.904,E2 -4239.904} C_VEL
LIN {X 0,Y 531.413,Z 252.171,A -85,B 0,C 180,E1 -4240.863,E2 -4240.863} C_VEL
LIN {X 0,Y 531.66,Z 240.493,A -85,B 0,C 180,E1 -4241.731,E2 -4241.731} C_VEL
LIN {X 0,Y 531.941,Z 229.01,A -85,B 0,C 180,E1 -4242.398,E2 -4242.398} C_VEL
LIN {X 0,Y 532.168,Z 217.003,A -85,B 0,C 180,E1 -4242.926,E2 -4242.926} C_VEL
LIN {X 0,Y 532.221,Z 206.687,A -85,B 0,C 180,E1 -4243.264,E2 -4243.264} C_VEL
LIN {X 0,Y 530.456,Z 197.141,A -85,B 0,C 180,E1 -4243.553,E2 -4243.553} C_VEL
LIN {X 0,Y 530.491,Z 192.637,A -85,B 0,C 180,E1 -4246.154,E2 -4246.154} C_VEL
LIN {X 0,Y 530.536,Z 188.538,A -85,B 0,C 180,E1 -4248.538,E2 -4248.538} C_VEL
LIN {X 0,Y 530.612,Z 184.429,A -85,B 0,C 180,E1 -4250.954,E2 -4250.954} C_VEL
LIN {X 0,Y 530.706,Z 179.419,A -85,B 0,C 180,E1 -4253.971,E2 -4253.971} C_VEL
LIN {X 0,Y 530.712,Z 174.906,A -85,B 0,C 180,E1 -4256.76,E2 -4256.76} C_VEL
LIN {X 0,Y 530.804,Z 170.816,A -85,B 0,C 180,E1 -4259.333,E2 -4259.333} C_VEL
LIN {X 0,Y 530.848,Z 166.527,A -85,B 0,C 180,E1 -4262.08,E2 -4262.08} C_VEL
LIN {X 0,Y 530.916,Z 162.282,A -85,B 0,C 180,E1 -4264.842,E2 -4264.842} C_VEL
LIN {X 0,Y 530.89,Z 161.357,A -85,B 0,C 180,E1 -4265.625,E2 -4265.625} C_VEL
LIN {X 0,Y 530.943,Z 161.351,A -85,B 0,C 180,E1 -4268.65,E2 -4268.65} C_VEL
LIN {X 0,Y 530.965,Z 161.345,A -85,B 0,C 180,E1 -4271.438,E2 -4271.438} C_VEL
LIN {X 0,Y 530.977,Z 161.343,A -85,B 0,C 180,E1 -4274.548,E2 -4274.548} C_VEL
LIN {X 0,Y 530.984,Z 161.341,A -85,B 0,C 180,E1 -4277.834,E2 -4277.834} C_VEL
LIN {X 0,Y 530.985,Z 161.345,A -85,B 0,C 180,E1 -4280.556,E2 -4280.556} C_VEL
LIN {X 0,Y 530.916,Z 161.35,A -85,B 0,C 180,E1 -4283.438,E2 -4283.438} C_VEL
LIN {X 0,Y 530.952,Z 161.348,A -85,B 0,C 180,E1 -4286.225,E2 -4286.225} C_VEL
LIN {X 0,Y 530.976,Z 161.346,A -85,B 0,C 180,E1 -4289.355,E2 -4289.355} C_VEL
LIN {X 0,Y 531.014,Z 161.342,A -85,B 0,C 180,E1 -4292.467,E2 -4292.467} C_VEL
LIN {X 0,Y 530.996,Z 161.339,A -85,B 0,C 180,E1 -4294.942,E2 -4294.942} C_VEL
LIN {X 0,Y 530.972,Z 161.345,A -85,B 0,C 180,E1 -4298.247,E2 -4298.247} C_VEL
LIN {X 0,Y 530.992,Z 161.342,A -85,B 0,C 180,E1 -4300.677,E2 -4300.677} C_VEL
LIN {X 0,Y 530.976,Z 161.347,A -85,B 0,C 180,E1 -4303.071,E2 -4303.071} C_VEL
LIN {X 0,Y 531.021,Z 161.337,A -85,B 0,C 180,E1 -4305.436,E2 -4305.436} C_VEL
LIN {X 0,Y 531.038,Z 161.336,A -85,B 0,C 180,E1 -4308.55,E2 -4308.55} C_VEL
LIN {X 0,Y 530.989,Z 161.345,A -85,B 0,C 180,E1 -4311.628,E2 -4311.628} C_VEL
LIN {X 0,Y 531.102,Z 161.33,A -85,B 0,C 180,E1 -4314.685,E2 -4314.685} C_VEL
LIN {X 0,Y 531.135,Z 161.324,A -85,B 0,C 180,E1 -4317.725,E2 -4317.725} C_VEL
LIN {X 0,Y 531.154,Z 161.321,A -85,B 0,C 180,E1 -4320.758,E2 -4320.758} C_VEL
LIN {X 0,Y 531.103,Z 161.328,A -85,B 0,C 180,E1 -4323.034,E2 -4323.034} C_VEL
LIN {X 0,Y 531.046,Z 161.333,A -85,B 0,C 180,E1 -4326.078,E2 -4326.078} C_VEL
LIN {X 0,Y 531.006,Z 161.339,A -85,B 0,C 180,E1 -4329.139,E2 -4329.139} C_VEL
LIN {X 0,Y 531.041,Z 161.339,A -85,B 0,C 180,E1 -4332.225,E2 -4332.225} C_VEL
LIN {X 0,Y 530.997,Z 161.344,A -85,B 0,C 180,E1 -4335.35,E2 -4335.35} C_VEL
LIN {X 0,Y 530.986,Z 161.344,A -85,B 0,C 180,E1 -4338.521,E2 -4338.521} C_VEL
LIN {X 0,Y 530.999,Z 161.341,A -85,B 0,C 180,E1 -4340.938,E2 -4340.938} C_VEL
LIN {X 0,Y 530.963,Z 161.348,A -85,B 0,C 180,E1 -4344.225,E2 -4344.225} C_VEL
LIN {X 0,Y 530.997,Z 161.34,A -85,B 0,C 180,E1 -4346.744,E2 -4346.744} C_VEL
LIN {X 0,Y 530.983,Z 161.347,A -85,B 0,C 180,E1 -4349.323,E2 -4349.323} C_VEL
LIN {X 0,Y 530.967,Z 161.345,A -85,B 0,C 180,E1 -4352.1,E2 -4352.1} C_VEL
LIN {X 0,Y 530.966,Z 161.345,A -85,B 0,C 180,E1 -4354.85,E2 -4354.85} C_VEL
LIN {X 0,Y 530.929,Z 161.352,A -85,B 0,C 180,E1 -4357.511,E2 -4357.511} C_VEL
LIN {X 0,Y 530.978,Z 161.342,A -85,B 0,C 180,E1 -4360.433,E2 -4360.433} C_VEL
LIN {X 0,Y 530.962,Z 161.346,A -85,B 0,C 180,E1 -4363.281,E2 -4363.281} C_VEL
LIN {X 0,Y 530.978,Z 161.343,A -85,B 0,C 180,E1 -4365.622,E2 -4365.622} C_VEL
LIN {X 0,Y 530.995,Z 161.342,A -85,B 0,C 180,E1 -4368.564,E2 -4368.564} C_VEL
LIN {X 0,Y 530.95,Z 161.352,A -85,B 0,C 180,E1 -4371.529,E2 -4371.529} C_VEL
LIN {X 0,Y 531.016,Z 161.48,A -85,B 0,C 180,E1 -4372.639,E2 -4372.639} C_VEL
LIN {X 0,Y 531.58,Z 165.661,A -85,B 0,C 180,E1 -4374.428,E2 -4374.428} C_VEL
LIN {X 0,Y 531.497,Z 172.404,A -85,B 0,C 180,E1 -4377.17,E2 -4377.17} C_VEL
LIN {X 0,Y 531.348,Z 180.317,A -85,B 0,C 180,E1 -4380.264,E2 -4380.264} C_VEL
LIN {X 0,Y 531.148,Z 188.108,A -85,B 0,C 180,E1 -4383.264,E2 -4383.264} C_VEL
LIN {X 0,Y 531.038,Z 195.243,A -85,B 0,C 180,E1 -4385.949,E2 -4385.949} C_VEL
LIN {X 0,Y 530.92,Z 202.578,A -85,B 0,C 180,E1 -4388.652,E2 -4388.652} C_VEL
LIN {X 0,Y 530.801,Z 209.256,A -85,B 0,C 180,E1 -4391.071,E2 -4391.071} C_VEL
LIN {X 0,Y 530.711,Z 217.048,A -85,B 0,C 180,E1 -4393.853,E2 -4393.853} C_VEL
LIN {X 0,Y 530.618,Z 224.491,A -85,B 0,C 180,E1 -4396.476,E2 -4396.476} C_VEL
LIN {X 0,Y 532.322,Z 235.263,A -85,B 0,C 180,E1 -4396.763,E2 -4396.763} C_VEL
LIN {X 0,Y 532.118,Z 247.766,A -85,B 0,C 180,E1 -4397.17,E2 -4397.17} C_VEL
LIN {X 0,Y 531.866,Z 259.408,A -85,B 0,C 180,E1 -4397.697,E2 -4397.697} C_VEL
LIN {X 0,Y 531.619,Z 270.592,A -85,B 0,C 180,E1 -4398.358,E2 -4398.358} C_VEL
LIN {X 0,Y 531.375,Z 282.259,A -85,B 0,C 180,E1 -4399.233,E2 -4399.233} C_VEL
LIN {X 0,Y 531.117,Z 291.537,A -85,B 0,C 180,E1 -4400.094,E2 -4400.094} C_VEL
LIN {X 0,Y 530.931,Z 299.99,A -85,B 0,C 180,E1 -4401.052,E2 -4401.052} C_VEL
LIN {X 0,Y 530.758,Z 308.236,A -85,B 0,C 180,E1 -4402.199,E2 -4402.199} C_VEL
LIN {X 0,Y 530.598,Z 315.269,A -85,B 0,C 180,E1 -4403.419,E2 -4403.419} C_VEL
LIN {X 0,Y 530.524,Z 320.949,A -85,B 0,C 180,E1 -4404.679,E2 -4404.679} C_VEL
LIN {X 0,Y 530.522,Z 324.895,A -85,B 0,C 180,E1 -4405.822,E2 -4405.822} C_VEL
LIN {X 0,Y 530.457,Z 327.808,A -85,B 0,C 180,E1 -4406.962,E2 -4406.962} C_VEL
LIN {X 0,Y 530.411,Z 329.197,A -85,B 0,C 180,E1 -4407.722,E2 -4407.722} C_VEL
LIN {X 0,Y 530.344,Z 330.785,A -85,B 0,C 180,E1 -4409.241,E2 -4409.241} C_VEL
LIN {X 0,Y 530.342,Z 331,A -85,B 0,C 180,E1 -4410,E2 -4410} C_VEL
LIN {X 0,Y 530.361,Z 330.186,A -85,B 0,C 180,E1 -4411.518,E2 -4411.518} C_VEL
LIN {X 0,Y 530.411,Z 329.199,A -85,B 0,C 180,E1 -4412.278,E2 -4412.278} C_VEL
LIN {X 0,Y 530.457,Z 327.81,A -85,B 0,C 180,E1 -4413.038,E2 -4413.038} C_VEL
LIN {X 0,Y 530.522,Z 324.896,A -85,B 0,C 180,E1 -4414.178,E2 -4414.178} C_VEL
LIN {X 0,Y 530.524,Z 320.95,A -85,B 0,C 180,E1 -4415.321,E2 -4415.321} C_VEL
LIN {X 0,Y 530.599,Z 315.262,A -85,B 0,C 180,E1 -4416.582,E2 -4416.582} C_VEL
LIN {X 0,Y 530.758,Z 308.239,A -85,B 0,C 180,E1 -4417.8,E2 -4417.8} C_VEL
LIN {X 0,Y 530.931,Z 299.992,A -85,B 0,C 180,E1 -4418.948,E2 -4418.948} C_VEL
LIN {X 0,Y 531.11,Z 291.541,A -85,B 0,C 180,E1 -4419.905,E2 -4419.905} C_VEL
LIN {X 0,Y 531.391,Z 281.101,A -85,B 0,C 180,E1 -4420.863,E2 -4420.863} C_VEL
LIN {X 0,Y 531.65,Z 269.29,A -85,B 0,C 180,E1 -4421.729,E2 -4421.729} C_VEL
LIN {X 0,Y 531.897,Z 257.491,A -85,B 0,C 180,E1 -4422.398,E2 -4422.398} C_VEL
LIN {X 0,Y 532.147,Z 245.177,A -85,B 0,C 180,E1 -4422.926,E2 -4422.926} C_VEL
LIN {X 0,Y 532.18,Z 233.899,A -85,B 0,C 180,E1 -4423.277,E2 -4423.277} C_VEL
LIN {X 0,Y 530.617,Z 224.492,A -85,B 0,C 180,E1 -4423.524,E2 -4423.524} C_VEL
LIN {X 0,Y 530.719,Z 215.936,A -85,B 0,C 180,E1 -4426.541,E2 -4426.541} C_VEL
LIN {X 0,Y 530.847,Z 208.144,A -85,B 0,C 180,E1 -4429.328,E2 -4429.328} C_VEL
LIN {X 0,Y 530.975,Z 200.519,A -85,B 0,C 180,E1 -4432.101,E2 -4432.101} C_VEL
LIN {X 0,Y 531.093,Z 192.562,A -85,B 0,C 180,E1 -4435.053,E2 -4435.053} C_VEL
LIN {X 0,Y 531.216,Z 184.77,A -85,B 0,C 180,E1 -4438.012,E2 -4438.012} C_VEL
LIN {X 0,Y 531.404,Z 177.763,A -85,B 0,C 180,E1 -4440.723,E2 -4440.723} C_VEL
LIN {X 0,Y 531.544,Z 170.15,A -85,B 0,C 180,E1 -4443.732,E2 -4443.732} C_VEL
LIN {X 0,Y 531.585,Z 165.644,A -85,B 0,C 180,E1 -4445.571,E2 -4445.571} C_VEL
LIN {X 0,Y 530.986,Z 161.346,A -85,B 0,C 180,E1 -4447.506,E2 -4447.506} C_VEL
LIN {X 0,Y 530.976,Z 161.349,A -85,B 0,C 180,E1 -4450.433,E2 -4450.433} C_VEL
LIN {X 0,Y 530.963,Z 161.346,A -85,B 0,C 180,E1 -4453.281,E2 -4453.281} C_VEL
LIN {X 0,Y 530.976,Z 161.346,A -85,B 0,C 180,E1 -4455.622,E2 -4455.622} C_VEL
LIN {X 0,Y 530.992,Z 161.343,A -85,B 0,C 180,E1 -4458.564,E2 -4458.564} C_VEL
LIN {X 0,Y 530.948,Z 161.345,A -85,B 0,C 180,E1 -4461.528,E2 -4461.528} C_VEL
LIN {X 0,Y 530.932,Z 161.35,A -85,B 0,C 180,E1 -4464.378,E2 -4464.378} C_VEL
LIN {X 0,Y 530.966,Z 161.347,A -85,B 0,C 180,E1 -4467.133,E2 -4467.133} C_VEL
LIN {X 0,Y 530.969,Z 161.344,A -85,B 0,C 180,E1 -4469.803,E2 -4469.803} C_VEL
LIN {X 0,Y 531.013,Z 161.343,A -85,B 0,C 180,E1 -4472.467,E2 -4472.467} C_VEL
LIN {X 0,Y 530.992,Z 161.34,A -85,B 0,C 180,E1 -4474.942,E2 -4474.942} C_VEL
LIN {X 0,Y 530.969,Z 161.344,A -85,B 0,C 180,E1 -4478.247,E2 -4478.247} C_VEL
LIN {X 0,Y 530.99,Z 161.342,A -85,B 0,C 180,E1 -4480.677,E2 -4480.677} C_VEL
LIN {X 0,Y 530.984,Z 161.346,A -85,B 0,C 180,E1 -4483.071,E2 -4483.071} C_VEL
LIN {X 0,Y 531.017,Z 161.338,A -85,B 0,C 180,E1 -4485.436,E2 -4485.436} C_VEL
LIN {X 0,Y 531.034,Z 161.336,A -85,B 0,C 180,E1 -4488.55,E2 -4488.55} C_VEL
LIN {X 0,Y 530.986,Z 161.344,A -85,B 0,C 180,E1 -4491.628,E2 -4491.628} C_VEL
LIN {X 0,Y 531.104,Z 161.33,A -85,B 0,C 180,E1 -4494.685,E2 -4494.685} C_VEL
LIN {X 0,Y 531.135,Z 161.324,A -85,B 0,C 180,E1 -4497.725,E2 -4497.725} C_VEL
LIN {X 0,Y 531.152,Z 161.321,A -85,B 0,C 180,E1 -4500.758,E2 -4500.758} C_VEL
LIN {X 0,Y 531.101,Z 161.33,A -85,B 0,C 180,E1 -4503.034,E2 -4503.034} C_VEL
LIN {X 0,Y 531.042,Z 161.334,A -85,B 0,C 180,E1 -4506.078,E2 -4506.078} C_VEL
LIN {X 0,Y 531.007,Z 161.338,A -85,B 0,C 180,E1 -4509.139,E2 -4509.139} C_VEL
LIN {X 0,Y 531.039,Z 161.338,A -85,B 0,C 180,E1 -4512.225,E2 -4512.225} C_VEL
LIN {X 0,Y 530.994,Z 161.344,A -85,B 0,C 180,E1 -4515.35,E2 -4515.35} C_VEL
LIN {X 0,Y 530.986,Z 161.345,A -85,B 0,C 180,E1 -4518.521,E2 -4518.521} C_VEL
LIN {X 0,Y 530.996,Z 161.342,A -85,B 0,C 180,E1 -4520.938,E2 -4520.938} C_VEL
LIN {X 0,Y 530.962,Z 161.346,A -85,B 0,C 180,E1 -4524.226,E2 -4524.226} C_VEL
LIN {X 0,Y 531.003,Z 161.339,A -85,B 0,C 180,E1 -4526.744,E2 -4526.744} C_VEL
LIN {X 0,Y 530.98,Z 161.346,A -85,B 0,C 180,E1 -4529.323,E2 -4529.323} C_VEL
LIN {X 0,Y 530.964,Z 161.346,A -85,B 0,C 180,E1 -4532.101,E2 -4532.101} C_VEL
LIN {X 0,Y 530.963,Z 161.345,A -85,B 0,C 180,E1 -4534.851,E2 -4534.851} C_VEL
LIN {X 0,Y 530.93,Z 161.353,A -85,B 0,C 180,E1 -4537.511,E2 -4537.511} C_VEL
LIN {X 0,Y 530.979,Z 161.341,A -85,B 0,C 180,E1 -4540.433,E2 -4540.433} C_VEL
LIN {X 0,Y 530.96,Z 161.346,A -85,B 0,C 180,E1 -4543.281,E2 -4543.281} C_VEL
LIN {X 0,Y 530.952,Z 161.345,A -85,B 0,C 180,E1 -4543.552,E2 -4543.552} C_VEL
LIN {X 0,Y 530.282,Z 161.431,A -85,B 0,C 180,E1 -4544.186,E2 -4544.186} C_VEL
LIN {X 0,Y 527.438,Z 161.784,A -85,B 0,C 180,E1 -4545.215,E2 -4545.215} C_VEL
LIN {X 0,Y 525.036,Z 162.086,A -85,B 0,C 180,E1 -4546.043,E2 -4546.043} C_VEL
LIN {X 0,Y 524.002,Z 162.214,A -85,B 0,C 180,E1 -4546.683,E2 -4546.683} C_VEL
LIN {X 0,Y 523.917,Z 162.223,A -85,B 0,C 180,E1 -4546.899,E2 -4546.899} C_VEL
LIN {X 0,Y 523.938,Z 162.223,A -85,B 0,C 180,E1 -4549.871,E2 -4549.871} C_VEL
LIN {X 0,Y 523.898,Z 162.228,A -85,B 0,C 180,E1 -4552.867,E2 -4552.867} C_VEL
LIN {X 0,Y 523.81,Z 162.429,A -85,B 0,C 180,E1 -4554.765,E2 -4554.765} C_VEL
LIN {X 0,Y 523.806,Z 166.871,A -85,B 0,C 180,E1 -4557.703,E2 -4557.703} C_VEL
LIN {X 0,Y 523.745,Z 171.522,A -85,B 0,C 180,E1 -4560.718,E2 -4560.718} C_VEL
LIN {X 0,Y 523.656,Z 176.239,A -85,B 0,C 180,E1 -4563.712,E2 -4563.712} C_VEL
LIN {X 0,Y 523.635,Z 180.318,A -85,B 0,C 180,E1 -4566.257,E2 -4566.257} C_VEL
LIN {X 0,Y 523.544,Z 184.394,A -85,B 0,C 180,E1 -4568.75,E2 -4568.75} C_VEL
LIN {X 0,Y 523.482,Z 188.5,A -85,B 0,C 180,E1 -4571.204,E2 -4571.204} C_VEL
LIN {X 0,Y 523.414,Z 192.638,A -85,B 0,C 180,E1 -4573.622,E2 -4573.622} C_VEL
LIN {X 0,Y 523.415,Z 197.506,A -85,B 0,C 180,E1 -4576.373,E2 -4576.373} C_VEL
LIN {X 0,Y 525.394,Z 208.913,A -85,B 0,C 180,E1 -4576.708,E2 -4576.708} C_VEL
LIN {X 0,Y 525.133,Z 222.162,A -85,B 0,C 180,E1 -4577.194,E2 -4577.194} C_VEL
LIN {X 0,Y 524.888,Z 234.344,A -85,B 0,C 180,E1 -4577.806,E2 -4577.806} C_VEL
LIN {X 0,Y 524.627,Z 245.084,A -85,B 0,C 180,E1 -4578.506,E2 -4578.506} C_VEL
LIN {X 0,Y 524.338,Z 255.78,A -85,B 0,C 180,E1 -4579.38,E2 -4579.38} C_VEL
LIN {X 0,Y 524.104,Z 265.4,A -85,B 0,C 180,E1 -4580.351,E2 -4580.351} C_VEL
LIN {X 0,Y 523.904,Z 273.28,A -85,B 0,C 180,E1 -4581.32,E2 -4581.32} C_VEL
LIN {X 0,Y 523.687,Z 280.986,A -85,B 0,C 180,E1 -4582.482,E2 -4582.482} C_VEL
LIN {X 0,Y 523.588,Z 288.05,A -85,B 0,C 180,E1 -4583.836,E2 -4583.836} C_VEL
LIN {X 0,Y 523.384,Z 292.763,A -85,B 0,C 180,E1 -4584.993,E2 -4584.993} C_VEL
LIN {X 0,Y 523.444,Z 296.367,A -85,B 0,C 180,E1 -4586.151,E2 -4586.151} C_VEL
LIN {X 0,Y 523.417,Z 298.232,A -85,B 0,C 180,E1 -4586.921,E2 -4586.921} C_VEL
LIN {X 0,Y 523.338,Z 299.641,A -85,B 0,C 180,E1 -4587.691,E2 -4587.691} C_VEL
LIN {X 0,Y 523.252,Z 301.259,A -85,B 0,C 180,E1 -4589.231,E2 -4589.231} C_VEL
LIN {X 0,Y 523.251,Z 301.497,A -85,B 0,C 180,E1 -4590,E2 -4590} C_VEL
LIN {X 0,Y 523.252,Z 301.315,A -85,B 0,C 180,E1 -4590.77,E2 -4590.77} C_VEL
LIN {X 0,Y 523.338,Z 299.768,A -85,B 0,C 180,E1 -4592.309,E2 -4592.309} C_VEL
LIN {X 0,Y 523.417,Z 298.413,A -85,B 0,C 180,E1 -4593.079,E2 -4593.079} C_VEL
LIN {X 0,Y 523.444,Z 295.554,A -85,B 0,C 180,E1 -4594.235,E2 -4594.235} C_VEL
LIN {X 0,Y 523.463,Z 291.676,A -85,B 0,C 180,E1 -4595.393,E2 -4595.393} C_VEL
LIN {X 0,Y 523.544,Z 286.448,A -85,B 0,C 180,E1 -4596.6,E2 -4596.6} C_VEL
LIN {X 0,Y 523.745,Z 279.15,A -85,B 0,C 180,E1 -4597.906,E2 -4597.906} C_VEL
LIN {X 0,Y 523.933,Z 271.006,A -85,B 0,C 180,E1 -4599.069,E2 -4599.069} C_VEL
LIN {X 0,Y 524.194,Z 262.668,A -85,B 0,C 180,E1 -4600.038,E2 -4600.038} C_VEL
LIN {X 0,Y 524.435,Z 252.377,A -85,B 0,C 180,E1 -4601.009,E2 -4601.009} C_VEL
LIN {X 0,Y 524.703,Z 241.17,A -85,B 0,C 180,E1 -4601.856,E2 -4601.856} C_VEL
LIN {X 0,Y 524.971,Z 231.023,A -85,B 0,C 180,E1 -4602.467,E2 -4602.467} C_VEL
LIN {X 0,Y 525.24,Z 218.497,A -85,B 0,C 180,E1 -4603.05,E2 -4603.05} C_VEL
LIN {X 0,Y 525.169,Z 206.881,A -85,B 0,C 180,E1 -4603.446,E2 -4603.446} C_VEL
LIN {X 0,Y 523.401,Z 197.357,A -85,B 0,C 180,E1 -4603.739,E2 -4603.739} C_VEL
LIN {X 0,Y 523.412,Z 192.794,A -85,B 0,C 180,E1 -4606.378,E2 -4606.378} C_VEL
LIN {X 0,Y 523.479,Z 188.657,A -85,B 0,C 180,E1 -4608.797,E2 -4608.797} C_VEL
LIN {X 0,Y 523.539,Z 184.543,A -85,B 0,C 180,E1 -4611.251,E2 -4611.251} C_VEL
LIN {X 0,Y 523.652,Z 179.847,A -85,B 0,C 180,E1 -4614.127,E2 -4614.127} C_VEL
LIN {X 0,Y 523.664,Z 175.019,A -85,B 0,C 180,E1 -4617.149,E2 -4617.149} C_VEL
LIN {X 0,Y 523.743,Z 170.912,A -85,B 0,C 180,E1 -4619.768,E2 -4619.768} C_VEL
LIN {X 0,Y 523.814,Z 166.771,A -85,B 0,C 180,E1 -4622.458,E2 -4622.458} C_VEL
LIN {X 0,Y 523.857,Z 162.572,A -85,B 0,C 180,E1 -4625.232,E2 -4625.232} C_VEL
LIN {X 0,Y 523.878,Z 162.232,A -85,B 0,C 180,E1 -4627.135,E2 -4627.135} C_VEL
LIN {X 0,Y 523.914,Z 162.226,A -85,B 0,C 180,E1 -4630.126,E2 -4630.126} C_VEL
LIN {X 0,Y 523.903,Z 162.224,A -85,B 0,C 180,E1 -4633.169,E2 -4633.169} C_VEL
LIN {X 0,Y 523.933,Z 162.222,A -85,B 0,C 180,E1 -4635.771,E2 -4635.771} C_VEL
LIN {X 0,Y 523.941,Z 162.224,A -85,B 0,C 180,E1 -4638.908,E2 -4638.908} C_VEL
LIN {X 0,Y 523.903,Z 162.224,A -85,B 0,C 180,E1 -4641.897,E2 -4641.897} C_VEL
LIN {X 0,Y 523.915,Z 162.223,A -85,B 0,C 180,E1 -4644.913,E2 -4644.913} C_VEL
LIN {X 0,Y 523.936,Z 162.223,A -85,B 0,C 180,E1 -4647.68,E2 -4647.68} C_VEL
LIN {X 0,Y 523.956,Z 162.221,A -85,B 0,C 180,E1 -4650.676,E2 -4650.676} C_VEL
LIN {X 0,Y 523.975,Z 162.214,A -85,B 0,C 180,E1 -4653.728,E2 -4653.728} C_VEL
LIN {X 0,Y 523.912,Z 162.226,A -85,B 0,C 180,E1 -4656.269,E2 -4656.269} C_VEL
LIN {X 0,Y 523.946,Z 162.218,A -85,B 0,C 180,E1 -4658.767,E2 -4658.767} C_VEL
LIN {X 0,Y 523.948,Z 162.222,A -85,B 0,C 180,E1 -4661.22,E2 -4661.22} C_VEL
LIN {X 0,Y 523.934,Z 162.221,A -85,B 0,C 180,E1 -4663.639,E2 -4663.639} C_VEL
LIN {X 0,Y 523.941,Z 162.222,A -85,B 0,C 180,E1 -4666.028,E2 -4666.028} C_VEL
LIN {X 0,Y 524.014,Z 162.212,A -85,B 0,C 180,E1 -4668.394,E2 -4668.394} C_VEL
LIN {X 0,Y 523.953,Z 162.223,A -85,B 0,C 180,E1 -4671.515,E2 -4671.515} C_VEL
LIN {X 0,Y 524.062,Z 162.206,A -85,B 0,C 180,E1 -4674.613,E2 -4674.613} C_VEL
LIN {X 0,Y 524.108,Z 162.199,A -85,B 0,C 180,E1 -4677.694,E2 -4677.694} C_VEL
LIN {X 0,Y 524.125,Z 162.197,A -85,B 0,C 180,E1 -4680.768,E2 -4680.768} C_VEL
LIN {X 0,Y 524.07,Z 162.205,A -85,B 0,C 180,E1 -4683.075,E2 -4683.075} C_VEL
LIN {X 0,Y 524.007,Z 162.21,A -85,B 0,C 180,E1 -4686.159,E2 -4686.159} C_VEL
LIN {X 0,Y 523.977,Z 162.214,A -85,B 0,C 180,E1 -4689.262,E2 -4689.262} C_VEL
LIN {X 0,Y 524.027,Z 162.211,A -85,B 0,C 180,E1 -4691.751,E2 -4691.751} C_VEL
LIN {X 0,Y 523.994,Z 162.215,A -85,B 0,C 180,E1 -4695.052,E2 -4695.052} C_VEL
LIN {X 0,Y 523.948,Z 162.218,A -85,B 0,C 180,E1 -4697.97,E2 -4697.97} C_VEL
LIN {X 0,Y 523.973,Z 162.219,A -85,B 0,C 180,E1 -4700.41,E2 -4700.41} C_VEL
LIN {X 0,Y 523.909,Z 162.222,A -85,B 0,C 180,E1 -4702.894,E2 -4702.894} C_VEL
LIN {X 0,Y 523.983,Z 162.217,A -85,B 0,C 180,E1 -4706.019,E2 -4706.019} C_VEL
LIN {X 0,Y 523.939,Z 162.223,A -85,B 0,C 180,E1 -4708.875,E2 -4708.875} C_VEL
LIN {X 0,Y 523.922,Z 162.222,A -85,B 0,C 180,E1 -4711.544,E2 -4711.544} C_VEL
LIN {X 0,Y 523.931,Z 162.224,A -85,B 0,C 180,E1 -4714.29,E2 -4714.29} C_VEL
LIN {X 0,Y 523.877,Z 162.233,A -85,B 0,C 180,E1 -4717.674,E2 -4717.674} C_VEL
LIN {X 0,Y 523.939,Z 162.218,A -85,B 0,C 180,E1 -4720.13,E2 -4720.13} C_VEL
LIN {X 0,Y 523.936,Z 162.221,A -85,B 0,C 180,E1 -4722.459,E2 -4722.459} C_VEL
LIN {X 0,Y 523.944,Z 162.219,A -85,B 0,C 180,E1 -4725.31,E2 -4725.31} C_VEL
LIN {X 0,Y 523.957,Z 162.218,A -85,B 0,C 180,E1 -4728.69,E2 -4728.69} C_VEL
LIN {X 0,Y 523.919,Z 162.227,A -85,B 0,C 180,E1 -4731.898,E2 -4731.898} C_VEL
LIN {X 0,Y 523.982,Z 162.348,A -85,B 0,C 180,E1 -4732.462,E2 -4732.462} C_VEL
LIN {X 0,Y 524.576,Z 166.699,A -85,B 0,C 180,E1 -4734.353,E2 -4734.353} C_VEL
LIN {X 0,Y 524.507,Z 173.442,A -85,B 0,C 180,E1 -4737.134,E2 -4737.134} C_VEL
LIN {X 0,Y 524.337,Z 180.228,A -85,B 0,C 180,E1 -4739.825,E2 -4739.825} C_VEL
LIN {X 0,Y 524.176,Z 188.108,A -85,B 0,C 180,E1 -4742.88,E2 -4742.88} C_VEL
LIN {X 0,Y 524.01,Z 195.719,A -85,B 0,C 180,E1 -4745.786,E2 -4745.786} C_VEL
LIN {X 0,Y 523.858,Z 203.691,A -85,B 0,C 180,E1 -4748.763,E2 -4748.763} C_VEL
LIN {X 0,Y 523.723,Z 211.482,A -85,B 0,C 180,E1 -4751.618,E2 -4751.618} C_VEL
LIN {X 0,Y 523.616,Z 219.274,A -85,B 0,C 180,E1 -4754.428,E2 -4754.428} C_VEL
LIN {X 0,Y 523.555,Z 224.491,A -85,B 0,C 180,E1 -4756.29,E2 -4756.29} C_VEL
LIN {X 0,Y 525.385,Z 236.177,A -85,B 0,C 180,E1 -4756.609,E2 -4756.609} C_VEL
LIN {X 0,Y 525.163,Z 248.981,A -85,B 0,C 180,E1 -4757.047,E2 -4757.047} C_VEL
LIN {X 0,Y 524.895,Z 261.173,A -85,B 0,C 180,E1 -4757.63,E2 -4757.63} C_VEL
LIN {X 0,Y 524.609,Z 272.267,A -85,B 0,C 180,E1 -4758.316,E2 -4758.316} C_VEL
LIN {X 0,Y 524.353,Z 283.399,A -85,B 0,C 180,E1 -4759.184,E2 -4759.184} C_VEL
LIN {X 0,Y 524.059,Z 293.334,A -85,B 0,C 180,E1 -4760.155,E2 -4760.155} C_VEL
LIN {X 0,Y 523.852,Z 302.959,A -85,B 0,C 180,E1 -4761.319,E2 -4761.319} C_VEL
LIN {X 0,Y 523.633,Z 310.62,A -85,B 0,C 180,E1 -4762.481,E2 -4762.481} C_VEL
LIN {X 0,Y 523.515,Z 317.679,A -85,B 0,C 180,E1 -4763.835,E2 -4763.835} C_VEL
LIN {X 0,Y 523.383,Z 322.372,A -85,B 0,C 180,E1 -4764.993,E2 -4764.993} C_VEL
LIN {X 0,Y 523.443,Z 325.957,A -85,B 0,C 180,E1 -4766.151,E2 -4766.151} C_VEL
LIN {X 0,Y 523.367,Z 327.807,A -85,B 0,C 180,E1 -4766.921,E2 -4766.921} C_VEL
LIN {X 0,Y 523.335,Z 329.197,A -85,B 0,C 180,E1 -4767.691,E2 -4767.691} C_VEL
LIN {X 0,Y 523.25,Z 330.785,A -85,B 0,C 180,E1 -4769.23,E2 -4769.23} C_VEL
LIN {X 0,Y 523.246,Z 331,A -85,B 0,C 180,E1 -4770,E2 -4770} C_VEL
LIN {X 0,Y 523.275,Z 330.186,A -85,B 0,C 180,E1 -4771.539,E2 -4771.539} C_VEL
LIN {X 0,Y 523.335,Z 329.199,A -85,B 0,C 180,E1 -4772.309,E2 -4772.309} C_VEL
LIN {X 0,Y 523.367,Z 327.81,A -85,B 0,C 180,E1 -4773.079,E2 -4773.079} C_VEL
LIN {X 0,Y 523.441,Z 324.896,A -85,B 0,C 180,E1 -4774.235,E2 -4774.235} C_VEL
LIN {X 0,Y 523.464,Z 320.949,A -85,B 0,C 180,E1 -4775.392,E2 -4775.392} C_VEL
LIN {X 0,Y 523.524,Z 315.724,A -85,B 0,C 180,E1 -4776.582,E2 -4776.582} C_VEL
LIN {X 0,Y 523.665,Z 309.469,A -85,B 0,C 180,E1 -4777.713,E2 -4777.713} C_VEL
LIN {X 0,Y 523.857,Z 301.48,A -85,B 0,C 180,E1 -4778.875,E2 -4778.875} C_VEL
LIN {X 0,Y 524.083,Z 293.337,A -85,B 0,C 180,E1 -4779.844,E2 -4779.844} C_VEL
LIN {X 0,Y 524.351,Z 283.403,A -85,B 0,C 180,E1 -4780.815,E2 -4780.815} C_VEL
LIN {X 0,Y 524.629,Z 272.237,A -85,B 0,C 180,E1 -4781.686,E2 -4781.686} C_VEL
LIN {X 0,Y 524.845,Z 261.18,A -85,B 0,C 180,E1 -4782.371,E2 -4782.371} C_VEL
LIN {X 0,Y 525.162,Z 248.984,A -85,B 0,C 180,E1 -4782.953,E2 -4782.953} C_VEL
LIN {X 0,Y 525.415,Z 236.185,A -85,B 0,C 180,E1 -4783.389,E2 -4783.389} C_VEL
LIN {X 0,Y 523.555,Z 224.492,A -85,B 0,C 180,E1 -4783.71,E2 -4783.71} C_VEL
LIN {X 0,Y 523.658,Z 215.936,A -85,B 0,C 180,E1 -4786.771,E2 -4786.771} C_VEL
LIN {X 0,Y 523.843,Z 206.794,A -85,B 0,C 180,E1 -4790.093,E2 -4790.093} C_VEL
LIN {X 0,Y 523.949,Z 199.24,A -85,B 0,C 180,E1 -4792.892,E2 -4792.892} C_VEL
LIN {X 0,Y 524.106,Z 190.902,A -85,B 0,C 180,E1 -4796.046,E2 -4796.046} C_VEL
LIN {X 0,Y 524.235,Z 183.648,A -85,B 0,C 180,E1 -4798.857,E2 -4798.857} C_VEL
LIN {X 0,Y 524.427,Z 176.809,A -85,B 0,C 180,E1 -4801.51,E2 -4801.51} C_VEL
LIN {X 0,Y 524.546,Z 170.061,A -85,B 0,C 180,E1 -4804.244,E2 -4804.244} C_VEL
LIN {X 0,Y 524.473,Z 165.547,A -85,B 0,C 180,E1 -4806.129,E2 -4806.129} C_VEL
LIN {X 0,Y 523.923,Z 162.226,A -85,B 0,C 180,E1 -4807.68,E2 -4807.68} C_VEL
LIN {X 0,Y 523.937,Z 162.225,A -85,B 0,C 180,E1 -4810.129,E2 -4810.129} C_VEL
LIN {X 0,Y 523.935,Z 162.222,A -85,B 0,C 180,E1 -4812.459,E2 -4812.459} C_VEL
LIN {X 0,Y 523.943,Z 162.223,A -85,B 0,C 180,E1 -4815.31,E2 -4815.31} C_VEL
LIN {X 0,Y 523.954,Z 162.222,A -85,B 0,C 180,E1 -4818.689,E2 -4818.689} C_VEL
LIN {X 0,Y 523.912,Z 162.222,A -85,B 0,C 180,E1 -4821.081,E2 -4821.081} C_VEL
LIN {X 0,Y 523.863,Z 162.231,A -85,B 0,C 180,E1 -4823.822,E2 -4823.822} C_VEL
LIN {X 0,Y 523.939,Z 162.219,A -85,B 0,C 180,E1 -4826.635,E2 -4826.635} C_VEL
LIN {X 0,Y 523.955,Z 162.221,A -85,B 0,C 180,E1 -4829.356,E2 -4829.356} C_VEL
LIN {X 0,Y 523.977,Z 162.218,A -85,B 0,C 180,E1 -4832.281,E2 -4832.281} C_VEL
LIN {X 0,Y 523.945,Z 162.22,A -85,B 0,C 180,E1 -4834.581,E2 -4834.581} C_VEL
LIN {X 0,Y 523.916,Z 162.228,A -85,B 0,C 180,E1 -4837.757,E2 -4837.757} C_VEL
LIN {X 0,Y 523.972,Z 162.215,A -85,B 0,C 180,E1 -4840.408,E2 -4840.408} C_VEL
LIN {X 0,Y 523.965,Z 162.22,A -85,B 0,C 180,E1 -4842.837,E2 -4842.837} C_VEL
LIN {X 0,Y 523.975,Z 162.216,A -85,B 0,C 180,E1 -4845.236,E2 -4845.236} C_VEL
LIN {X 0,Y 524.011,Z 162.212,A -85,B 0,C 180,E1 -4848.394,E2 -4848.394} C_VEL
LIN {X 0,Y 523.95,Z 162.222,A -85,B 0,C 180,E1 -4851.515,E2 -4851.515} C_VEL
LIN {X 0,Y 524.064,Z 162.206,A -85,B 0,C 180,E1 -4854.613,E2 -4854.613} C_VEL
LIN {X 0,Y 524.108,Z 162.199,A -85,B 0,C 180,E1 -4857.694,E2 -4857.694} C_VEL
LIN {X 0,Y 524.122,Z 162.197,A -85,B 0,C 180,E1 -4860.768,E2 -4860.768} C_VEL
LIN {X 0,Y 524.067,Z 162.206,A -85,B 0,C 180,E1 -4863.075,E2 -4863.075} C_VEL
LIN {X 0,Y 524.003,Z 162.211,A -85,B 0,C 180,E1 -4866.16,E2 -4866.16} C_VEL
LIN {X 0,Y 523.978,Z 162.213,A -85,B 0,C 180,E1 -4869.262,E2 -4869.262} C_VEL
LIN {X 0,Y 524.001,Z 162.214,A -85,B 0,C 180,E1 -4871.739,E2 -4871.739} C_VEL
LIN {X 0,Y 523.991,Z 162.216,A -85,B 0,C 180,E1 -4875.053,E2 -4875.053} C_VEL
LIN {X 0,Y 523.962,Z 162.217,A -85,B 0,C 180,E1 -4877.969,E2 -4877.969} C_VEL
LIN {X 0,Y 523.97,Z 162.221,A -85,B 0,C 180,E1 -4880.41,E2 -4880.41} C_VEL
LIN {X 0,Y 523.906,Z 162.223,A -85,B 0,C 180,E1 -4882.894,E2 -4882.894} C_VEL
LIN {X 0,Y 523.983,Z 162.215,A -85,B 0,C 180,E1 -4886.02,E2 -4886.02} C_VEL
LIN {X 0,Y 523.938,Z 162.222,A -85,B 0,C 180,E1 -4888.875,E2 -4888.875} C_VEL
LIN {X 0,Y 523.92,Z 162.222,A -85,B 0,C 180,E1 -4891.544,E2 -4891.544} C_VEL
LIN {X 0,Y 523.928,Z 162.224,A -85,B 0,C 180,E1 -4894.291,E2 -4894.291} C_VEL
LIN {X 0,Y 523.878,Z 162.231,A -85,B 0,C 180,E1 -4897.674,E2 -4897.674} C_VEL
LIN {X 0,Y 523.937,Z 162.218,A -85,B 0,C 180,E1 -4900.13,E2 -4900.13} C_VEL
LIN {X 0,Y 523.934,Z 162.221,A -85,B 0,C 180,E1 -4902.459,E2 -4902.459} C_VEL
LIN {X 0,Y 523.954,Z 162.217,A -85,B 0,C 180,E1 -4905.309,E2 -4905.309} C_VEL
LIN {X 0,Y 523.917,Z 162.223,A -85,B 0,C 180,E1 -4906.899,E2 -4906.899} C_VEL
LIN {X 0,Y 523.246,Z 162.308,A -85,B 0,C 180,E1 -4907.541,E2 -4907.541} C_VEL
LIN {X 0,Y 520.39,Z 162.663,A -85,B 0,C 180,E1 -4908.582,E2 -4908.582} C_VEL
LIN {X 0,Y 517.979,Z 162.966,A -85,B 0,C 180,E1 -4909.421,E2 -4909.421} C_VEL
LIN {X 0,Y 516.944,Z 163.093,A -85,B 0,C 180,E1 -4910.069,E2 -4910.069} C_VEL
LIN {X 0,Y 516.861,Z 163.102,A -85,B 0,C 180,E1 -4910.288,E2 -4910.288} C_VEL
LIN {X 0,Y 516.844,Z 163.109,A -85,B 0,C 180,E1 -4913.252,E2 -4913.252} C_VEL
LIN {X 0,Y 516.754,Z 163.204,A -85,B 0,C 180,E1 -4914.688,E2 -4914.688} C_VEL
LIN {X 0,Y 516.75,Z 167.368,A -85,B 0,C 180,E1 -4917.483,E2 -4917.483} C_VEL
LIN {X 0,Y 516.705,Z 172.245,A -85,B 0,C 180,E1 -4920.682,E2 -4920.682} C_VEL
LIN {X 0,Y 516.599,Z 177.233,A -85,B 0,C 180,E1 -4923.882,E2 -4923.882} C_VEL
